(* CODESYS project plc_chalet_xts.library
   Title: CHALET_Xts
   Version: 1.7.6
   Placeholder: CHALET_Xts
   Company: Beckhoff CH

Project tree, tasks and I/O mapping:
  libraries: CHALET_BaseComponents, * (Beckhoff CH); CHALET_Nc, * (Beckhoff CH); Tc2_EtherCAT, * (Beckhoff Automation GmbH); Tc2_Math, * (Beckhoff Automation GmbH); Tc2_MC2, * (Beckhoff Automation GmbH); Tc2_Standard, * (Beckhoff Automation GmbH); Tc2_System, * (Beckhoff Automation GmbH); Tc3_Mc3Definitions, * (Beckhoff Automation GmbH); Tc3_McCollisionAvoidance, * (Beckhoff Automation GmbH); Tc3_McCoordinatedMotion, * (Beckhoff Automation GmbH); Tc3_Module, * (Beckhoff Automation GmbH); Tc3_XTS_Utility, * (Beckhoff Automation GmbH)
  COMPENENTs/
    Casting/
      function ToEnvironment [ST]
      function ToGroup [ST]
      function ToMover [ST]
      function ToMover_PLC [ST]
      function ToStation [ST]
      function ToStation_PLC [ST]
      function ToTrigger [ST]
    Environment/
      function block FB_XTS_Environment [ST]: FB_init, HR, Initialize, TrackIsRing, TrackLength, Update, UtilityEnvirement
      interface I_XTS_Environment: HR, Initialize, TrackIsRing, TrackLength, Update, UtilityEnvirement
    Group/
      data type E_NcGroupCommands
      function block FB_XTS_Group [ST]: AddAxisListToGroup, AddingAxisToGroup, AllAxesStanding, ChangeGapMode, Disable, Enable, FB_init, GroupEnabled, HR, Initialize, OID, RemoveAxisFromGroup, Reset, UngroupAllAxes, Update, UtilityCAGroup
      interface I_XTS_Group: AddAxisListToGroup, AddingAxisToGroup, AllAxesStanding, ChangeGapMode, Disable, Enable, GroupEnabled, HR, Initialize, RemoveAxisFromGroup, Reset, UngroupAllAxes, Update, UtilityCAGroup
    Mover/
      function block FB_XTS_Axis [ST]: HaltCA, MoveAbsoluteCA, Update
      function block FB_XTS_Mover [ST]: Disable, Enable, HaltCA, MoveAbsCA, Reset, Coupled, DrivenDistance, Feedback, Gap, getAxisRef, IdentInGroup, LagDistance, MoveAbsPosition, MoveAbsVelocity, MoverInGroup, Moving, NextMover, OID, ParentStation, PositionOnTrack, SetAcceleration, SetVelocity, TargedStation, FB_init, Initialize, Update, UtilityMover
      interface I_XTS_Mover: Coupled, Disable, DrivenDistance, Enable, Feedback, Gap, getAxisRef, HaltCA, IdentInGroup, LagDistance, MoveAbsCA, MoveAbsPosition, MoveAbsVelocity, MoverInGroup, Moving, NextMover, OID, ParentStation, PositionOnTrack, Reset, SetAcceleration, SetVelocity, TargedStation, UtilityMover
      interface I_XTS_Mover_PLC: DrivenDistance, Gap, LagDistance, PositionOnTrack, SetVelocity, TargedStation, UtilityMover
    Station/
      data type E_Colors_ARGB
      function block FB_XTS_Station [ST]: AddMoverToQueue, AreMoversInPlace, CtsEmptySpaceInQueue, CtsMoversInQueue, DeleteMoversQueue, FB_init, HR, Initialize, LUID, MoverGapAtExit, MoverQueueSize, MoversInQueue, MoverVelocityAtExit, OID, PositionOnTrack, SendMoversToStation, StationBehinde, StationGroupID, StationInFront, SuppressDynamicsChange, TrySendMoverToNextStation, Update, UtilityStationInfo
      interface I_XTS_Station: AddMoverToQueue, AreMoversInPlace, CtsEmptySpaceInQueue, CtsMoversInQueue, DeleteMoversQueue, HR, MoverGapAtExit, MoverQueueSize, MoversInQueue, MoverVelocityAtExit, PositionOnTrack, SendMoversToStation, StationGroupID, StationInFront
      interface I_XTS_Station_PLC: AreMoversInPlace, MoverQueueSize, MoversInQueue, SendMoversToStation, SuppressDynamicsChange
    System/
      function block FB_XTS_System [ST]: Disable, Disabled, Disabling, Enable, Enabled, Enabling, Environment, Feedback, getMoverInFront, getStationInFront, Initialize, Initialized, LinkEnvironment, LinkGroup, Movers, RegisterMover, RegisterStation, RegisterTrigger, RegisterZone, Reset, Station, Stations, SuppressAllDynamicsChanges, TrackLength, Update
      interface I_XTS_System_PLC: Disable, Disabled, Enable, Enabled, Feedback, Initialize, Initialized, Reset, Station, SuppressAllDynamicsChanges, TrackLength, Update
      interface I_XTS_System_Registration: Disabled, Enabled, Environment, getMoverInFront, getStationInFront, Initialized, LinkEnvironment, LinkGroup, Movers, RegisterMover, RegisterStation, RegisterTrigger, RegisterZone, Stations, TrackLength
    Trigger/
      function block FB_XTS_Trigger [ST]: FB_init, HR, Initialize, ListOfMoversToCheck, MoverAtTrigger, MoverDetected, PositionOnTrack, Prepare, TimeStamp, TriggerDirection, Update
      interface I_XTS_Trigger: HR, ListOfMoversToCheck, MoverAtTrigger, MoverDetected, PositionOnTrack, TimeStamp, TriggerDirection
    Zone/
      function block FB_XTS_Zone [ST]: CtsMoversInZone, EndPositionOnTrack, FB_init, HR, Initialize, ListOfMoversToCheck, MoversInZone, Prepare, StartPositionOnTrack, Update
      interface I_XTS_Zone: CtsMoversInZone, EndPositionOnTrack, HR, ListOfMoversToCheck, MoversInZone, StartPositionOnTrack
    Class Diagram
  FUNCTIONs/
    function FUN_BuildLogString [ST]
    function FUN_GetDistToPosModulo [ST]
    function FUN_InLimitTest [ST]
  00000000-0000-0000-0000-000000000000|Disclaimer Standard DE R1006.pdf
  Disclaimer Standard DE R1006.pdf
  global variables XtsParameterlist
*)

// COMPENENTs/Group/E_NcGroupCommands
{attribute 'qualified_only'}
{attribute 'strict'}
{attribute 'to_string'}
TYPE E_NcGroupCommands :
(
	None:=0,
	GroupDisable:=150,
	GroupEnable,
	GroupReset,
	AddAxisListToGroup,
	RemoveAxisFromGroup,
	UngroupAllAxes
);
END_TYPE

// COMPENENTs/Station/E_Colors_ARGB
{attribute 'qualified_only'}
{attribute 'strict'}
{attribute 'to_string'}
TYPE E_Colors_ARGB : (
        Darkred              := 16#FF8B0000, // rgb(139,0,0)
        Brown                := 16#FFA52A2A, // rgb(165,42,42)
        Firebrick            := 16#FFB22222, // rgb(178,34,34)
        Crimson              := 16#FFDC143C, // rgb(220,20,60)
        Red                  := 16#FFFF0000, // rgb(255,0,0)
        Tomato               := 16#FFFF6347, // rgb(255,99,71)
        Coral                := 16#FFFF7F50, // rgb(255,127,80)
        Indianred            := 16#FFCD5C5C, // rgb(205,92,92)
        Lightcoral           := 16#FFF08080, // rgb(240,128,128)
        Darksalmon           := 16#FFE9967A, // rgb(233,150,122)
        Salmon               := 16#FFFA8072, // rgb(250,128,114)
        Lightsalmon          := 16#FFFFA07A, // rgb(255,160,122)
        Orangered            := 16#FFFF4500, // rgb(255,69,0)
        Darkorange           := 16#FFFF8C00, // rgb(255,140,0)
        Orange               := 16#FFFFA500, // rgb(255,165,0)
        Gold                 := 16#FFFFD700, // rgb(255,215,0)
        Darkgoldenrod        := 16#FFB8860B, // rgb(184,134,11)
        Goldenrod            := 16#FFDAA520, // rgb(218,165,32)
        Palegoldenrod        := 16#FFEEE8AA, // rgb(238,232,170)
        Darkkhaki            := 16#FFBDB76B, // rgb(189,183,107)
        Khaki                := 16#FFF0E68C, // rgb(240,230,140)
        Olive                := 16#FF808000, // rgb(128,128,0)
        Yellow               := 16#FFFFFF00, // rgb(255,255,0)
        Yellowgreen          := 16#FF9ACD32, // rgb(154,205,50)
        Darkolivegreen       := 16#FF556B2F, // rgb(85,107,47)
        Olivedrab            := 16#FF6B8E23, // rgb(107,142,35)
        Lawngreen            := 16#FF7CFC00, // rgb(124,252,0)
        Chartreuse           := 16#FF7FFF00, // rgb(127,255,0)
        Greenyellow          := 16#FFADFF2F, // rgb(173,255,47)
        Darkgreen            := 16#FF006400, // rgb(0,100,0)
        Green                := 16#FF008000, // rgb(0,128,0)
        Forestgreen          := 16#FF228B22, // rgb(34,139,34)
        Lime                 := 16#FF00FF00, // rgb(0,255,0)
        Limegreen            := 16#FF32CD32, // rgb(50,205,50)
        Lightgreen           := 16#FF90EE90, // rgb(144,238,144)
        Palegreen            := 16#FF98FB98, // rgb(152,251,152)
        Darkseagreen         := 16#FF8FBC8F, // rgb(143,188,143)
        Mediumspringgreen    := 16#FF00FA9A, // rgb(0,250,154)
        Springgreen          := 16#FF00FF7F, // rgb(0,255,127)
        Seagreen             := 16#FF2E8B57, // rgb(46,139,87)
        Mediumaquamarine     := 16#FF66CDAA, // rgb(102,205,170)
        Mediumseagreen       := 16#FF3CB371, // rgb(60,179,113)
        Lightseagreen        := 16#FF20B2AA, // rgb(32,178,170)
        Darkslategray        := 16#FF2F4F4F, // rgb(47,79,79)
        Teal                 := 16#FF008080, // rgb(0,128,128)
        Darkcyan             := 16#FF008B8B, // rgb(0,139,139)
        Aqua                 := 16#FF00FFFF, // rgb(0,255,255)
        Lightcyan            := 16#FFE0FFFF, // rgb(224,255,255)
        Darkturquoise        := 16#FF00CED1, // rgb(0,206,209)
        Turquoise            := 16#FF40E0D0, // rgb(64,224,208)
        Mediumturquoise      := 16#FF48D1CC, // rgb(72,209,204)
        Paleturquoise        := 16#FFAFEEEE, // rgb(175,238,238)
        Aquamarine           := 16#FF7FFFD4, // rgb(127,255,212)
        Powderblue           := 16#FFB0E0E6, // rgb(176,224,230)
        Cadetblue            := 16#FF5F9EA0, // rgb(95,158,160)
        Steelblue            := 16#FF4682B4, // rgb(70,130,180)
        Cornflowerblue       := 16#FF6495ED, // rgb(100,149,237)
        Deepskyblue          := 16#FF00BFFF, // rgb(0,191,255)
        Dodgerblue           := 16#FF1E90FF, // rgb(30,144,255)
        Lightblue            := 16#FFADD8E6, // rgb(173,216,230)
        Skyblue              := 16#FF87CEEB, // rgb(135,206,235)
        Lightskyblue         := 16#FF87CEFA, // rgb(135,206,250)
        Midnightblue         := 16#FF191970, // rgb(25,25,112)
        Navy                 := 16#FF000080, // rgb(0,0,128)
        Darkblue             := 16#FF00008B, // rgb(0,0,139)
        Mediumblue           := 16#FF0000CD, // rgb(0,0,205)
        Blue                 := 16#FF0000FF, // rgb(0,0,255)
        Royalblue            := 16#FF4169E1, // rgb(65,105,225)
        Blueviolet           := 16#FF8A2BE2, // rgb(138,43,226)
        Indigo               := 16#FF4B0082, // rgb(75,0,130)
        Darkslateblue        := 16#FF483D8B, // rgb(72,61,139)
        Slateblue            := 16#FF6A5ACD, // rgb(106,90,205)
        Mediumslateblue      := 16#FF7B68EE, // rgb(123,104,238)
        Mediumpurple         := 16#FF9370DB, // rgb(147,112,219)
        Darkmagenta          := 16#FF8B008B, // rgb(139,0,139)
        Darkviolet           := 16#FF9400D3, // rgb(148,0,211)
        Darkorchid           := 16#FF9932CC, // rgb(153,50,204)
        Mediumorchid         := 16#FFBA55D3, // rgb(186,85,211)
        Purple               := 16#FF800080, // rgb(128,0,128)
        Thistle              := 16#FFD8BFD8, // rgb(216,191,216)
        Plum                 := 16#FFDDA0DD, // rgb(221,160,221)
        Violet               := 16#FFEE82EE, // rgb(238,130,238)
        Magenta              := 16#FFFF00FF, // rgb(255,0,255)
        Orchid               := 16#FFDA70D6, // rgb(218,112,214)
        Mediumvioletred      := 16#FFC71585, // rgb(199,21,133)
        Palevioletred        := 16#FFDB7093, // rgb(219,112,147)
        Deeppink             := 16#FFFF1493, // rgb(255,20,147)
        Hotpink              := 16#FFFF69B4, // rgb(255,105,180)
        Lightpink            := 16#FFFFB6C1, // rgb(255,182,193)
        Pink                 := 16#FFFFC0CB, // rgb(255,192,203)
        Antiquewhite         := 16#FFFAEBD7, // rgb(250,235,215)
        Beige                := 16#FFF5F5DC, // rgb(245,245,220)
        Bisque               := 16#FFFFE4C4, // rgb(255,228,196)
        Blanchedalmond       := 16#FFFFEBCD, // rgb(255,235,205)
        Wheat                := 16#FFF5DEB3, // rgb(245,222,179)
        Cornsilk             := 16#FFFFF8DC, // rgb(255,248,220)
        Lemonchiffon         := 16#FFFFFACD, // rgb(255,250,205)
        LightGoldenRodYellow := 16#FFFAFAD2, // rgb(250,250,210)
        LightYellow          := 16#FFFFFFE0, // rgb(255,255,224)
        SaddleBrown          := 16#FF8B4513, // rgb(139,69,19)
        Sienna               := 16#FFA0522D, // rgb(160,82,45)
        Chocolate            := 16#FFD2691E, // rgb(210,105,30)
        Peru                 := 16#FFCD853F, // rgb(205,133,63)
        SandyBrown           := 16#FFF4A460, // rgb(244,164,96)
        BurlyWood            := 16#FFDEB887, // rgb(222,184,135)
        RosyBrown            := 16#FFBC8F8F, // rgb(188,143,143)
        Moccasin             := 16#FFFFE4B5, // rgb(255,228,181)
        NavajoWhite          := 16#FFFFDEAD, // rgb(255,222,173)
        PeachPuff            := 16#FFFFDAB9, // rgb(255,218,185)
        MistyRose            := 16#FFFFE4E1, // rgb(255,228,225)
        LavenderBlush        := 16#FFFFF0F5, // rgb(255,240,245)
        Linen                := 16#FFFAF0E6, // rgb(250,240,230)
        OldLace              := 16#FFFDF5E6, // rgb(253,245,230)
        PapayaWhip           := 16#FFFFEFD5, // rgb(255,239,213)
        Seashell             := 16#FFFFF5EE, // rgb(255,245,238)
        MintCream            := 16#FFF5FFFA, // rgb(245,255,250)
        SlateGray            := 16#FF708090, // rgb(112,128,144)
        LightSlateGray       := 16#FF778899, // rgb(119,136,153)
        LightSteelBlue       := 16#FFB0C4DE, // rgb(176,196,222)
        Lavender             := 16#FFE6E6FA, // rgb(230,230,250)
        FloralWhite          := 16#FFFFFAF0, // rgb(255,250,240)
        AliceBlue            := 16#FFF0F8FF, // rgb(240,248,255)
        GhostWhite           := 16#FFF8F8FF, // rgb(248,248,255)
        HoneyDew             := 16#FFF0FFF0, // rgb(240,255,240)
        Ivory                := 16#FFFFFFF0, // rgb(255,255,240)
        Azure                := 16#FFF0FFFF, // rgb(240,255,255)
        Snow                 := 16#FFFFFAFA, // rgb(255,250,250)
        Black                := 16#FF000000, // rgb(0,0,0)
        DimGray              := 16#FF696969, // rgb(105,105,105)
        Gray                 := 16#FF808080, // rgb(128,128,128)
        DarkGray             := 16#FFA9A9A9, // rgb(169,169,169)
        Silver               := 16#FFC0C0C0, // rgb(192,192,192)
        LightGray            := 16#FFD3D3D3, // rgb(211,211,211)
        Gainsboro            := 16#FFDCDCDC, // rgb(220,220,220)
        WhiteSmoke           := 16#FFF5F5F5, // rgb(245,245,245)
        White                := 16#FFFFFFFF  // rgb(255,255,255)
    ) UDINT;
END_TYPE

// XtsParameterlist
{attribute 'qualified_only'}
VAR_GLOBAL CONSTANT
	MAX_MOVER_PER_SYSTEM : UINT := 50;
END_VAR

// COMPENENTs/Casting/ToEnvironment
FUNCTION ToEnvironment : BOOL
VAR_INPUT
	iChObject : I_CH_OBJECT;
	iXtsEnvironment : REFERENCE TO I_XTS_Environment;
END_VAR

VAR
	iTmp : I_XTS_Environment;
END_VAR

(* 
   1. Test if the interface exists
   2. Test if the object implements a "Object" interface 
   3. Write reference to interface in parameter
   4. Returne TRUE if succesfull
*)
IF iChObject <> 0 AND_THEN __QUERYINTERFACE(iChObject,iTmp) THEN
	iXtsEnvironment := iTmp;
	ToEnvironment := TRUE;
END_IF

END_FUNCTION

// COMPENENTs/Environment/I_XTS_Environment
INTERFACE I_XTS_Environment  EXTENDS __SYSTEM.IQueryInterface

{attribute 'monitoring':='call'}
PROPERTY HR : HRESULT
GET
END_GET
END_PROPERTY

METHOD Initialize : HRESULT
END_METHOD

{attribute 'monitoring':='call'}
PROPERTY TrackIsRing : BOOL
GET
END_GET
END_PROPERTY

{attribute 'monitoring':='call'}
PROPERTY TrackLength : LREAL
GET
END_GET
END_PROPERTY

METHOD Update : HRESULT
VAR_INPUT
END_VAR
END_METHOD

PROPERTY UtilityEnvirement : Tc3_XTS_Utility.i_TcIoXtsEnvironment
GET
END_GET
END_PROPERTY

END_INTERFACE

// COMPENENTs/Casting/ToGroup
FUNCTION ToGroup : BOOL
VAR_INPUT
	iChObject : I_CH_OBJECT;
	iXtsGroup : REFERENCE TO I_XTS_Group;
END_VAR

VAR
	iTmp : I_XTS_Group;
END_VAR

(* 
   1. Test if the interface exists
   2. Test if the object implements a "Object" interface 
   3. Write reference to interface in parameter
   4. Returne TRUE if succesfull
*)
IF iChObject <> 0 AND_THEN __QUERYINTERFACE(iChObject,iTmp) THEN
	iXtsGroup := iTmp;
	ToGroup := TRUE;
END_IF

END_FUNCTION

// COMPENENTs/Group/I_XTS_Group
INTERFACE I_XTS_Group  EXTENDS __SYSTEM.IQueryInterface

METHOD AddAxisListToGroup : HRESULT
VAR_INPUT
	iMovers : I_CH_List;
END_VAR
END_METHOD

METHOD AddingAxisToGroup : HRESULT
END_METHOD

PROPERTY AllAxesStanding : Bool
GET
END_GET
END_PROPERTY

METHOD ChangeGapMode : HRESULT
VAR_INPUT
	bFast : BOOL;
END_VAR
END_METHOD

METHOD Disable : HRESULT
VAR_INPUT
END_VAR
END_METHOD

METHOD Enable : HRESULT
VAR_INPUT
END_VAR
END_METHOD

{attribute 'monitoring':='call'}
PROPERTY GroupEnabled : BOOL
GET
END_GET
END_PROPERTY

{attribute 'monitoring':='call'}
PROPERTY HR : HRESULT
GET
END_GET
END_PROPERTY

METHOD Initialize : HRESULT
VAR_INPUT
END_VAR
END_METHOD

METHOD RemoveAxisFromGroup : HRESULT
VAR_INPUT
	iMover : I_XTS_Mover;
END_VAR
END_METHOD

METHOD Reset : HRESULT
VAR_INPUT
END_VAR
END_METHOD

METHOD UngroupAllAxes : HRESULT
VAR_INPUT
END_VAR
END_METHOD

METHOD Update : HRESULT
VAR_INPUT
END_VAR
END_METHOD

{attribute 'monitoring':='call'}
PROPERTY UtilityCAGroup : I_Mc2CaGroup
GET
END_GET
END_PROPERTY

END_INTERFACE

// COMPENENTs/Mover/I_XTS_Mover
INTERFACE I_XTS_Mover EXTENDS __SYSTEM.IQueryInterface

{attribute 'OPC.UA.DA.Property' := '1'}
{attribute 'monitoring':='call'}
PROPERTY Coupled : BOOL
GET
END_GET
END_PROPERTY

METHOD Disable : HRESULT
VAR_INPUT
END_VAR
END_METHOD

{attribute 'monitoring':='call'}
PROPERTY DrivenDistance : LREAL
GET
END_GET
END_PROPERTY

METHOD Enable : HRESULT
VAR_INPUT
END_VAR
END_METHOD

{attribute 'OPC.UA.DA.Property' := '1'}
{attribute 'monitoring':='call'}
PROPERTY Feedback : I_CH_Feedback
GET
END_GET
END_PROPERTY

{attribute 'monitoring':='call'}
PROPERTY Gap : LREAL
GET
END_GET
END_PROPERTY

PROPERTY getAxisRef : REFERENCE TO Tc2_MC2.AXIS_REF
GET
END_GET
END_PROPERTY

METHOD HaltCA : HRESULT
VAR_INPUT
END_VAR
END_METHOD

{attribute 'monitoring':='call'}
PROPERTY IdentInGroup : IDENT_IN_GROUP_REF
GET
END_GET
END_PROPERTY

{attribute 'monitoring':='call'}
PROPERTY LagDistance : LREAL
GET
END_GET
END_PROPERTY

METHOD MoveAbsCA : HRESULT
VAR_INPUT
    Position              : MC_LREAL := MC_INVALID;
    Velocity              : MC_LREAL := MC_INVALID;
    Gap                   : MC_LREAL := MC_DEFAULT;
    Direction             : Tc3_Mc3Definitions.MC_DIRECTION;
END_VAR
END_METHOD

{attribute 'monitoring':='call'}
PROPERTY MoveAbsPosition : LREAL
GET
END_GET
END_PROPERTY

{attribute 'monitoring':='call'}
PROPERTY MoveAbsVelocity : LREAL
GET
END_GET
END_PROPERTY

PROPERTY MoverInGroup : Bool
GET
END_GET
SET
END_SET
END_PROPERTY

{attribute 'OPC.UA.DA.Property' := '1'}
{attribute 'monitoring':='call'}
PROPERTY Moving : BOOL
GET
END_GET
END_PROPERTY

{attribute 'monitoring':='call'}
PROPERTY NextMover : I_XTS_Mover
GET
END_GET
END_PROPERTY

PROPERTY OID : OTCID
GET
END_GET
END_PROPERTY

{attribute 'monitoring':='call'}
PROPERTY ParentStation : I_XTS_Station
GET
END_GET
SET
END_SET
END_PROPERTY

{attribute 'monitoring':='call'}
PROPERTY PositionOnTrack : LREAL
GET
END_GET
END_PROPERTY

METHOD Reset : HRESULT
VAR_INPUT
END_VAR
END_METHOD

{attribute 'monitoring':='call'}
PROPERTY SetAcceleration : LREAL
GET
END_GET
END_PROPERTY

{attribute 'monitoring':='call'}
PROPERTY SetVelocity : LREAL
GET
END_GET
END_PROPERTY

{attribute 'monitoring':='call'}
PROPERTY TargedStation : STRING
GET
END_GET
SET
END_SET
END_PROPERTY

{attribute 'monitoring':='call'}
PROPERTY UtilityMover : I_TcIoXtsXpuMover
GET
END_GET
END_PROPERTY

END_INTERFACE

// COMPENENTs/Station/I_XTS_Station
INTERFACE I_XTS_Station  EXTENDS __SYSTEM.IQueryInterface

METHOD AddMoverToQueue : HRESULT
VAR_INPUT
	iMover : I_XTS_Mover;
END_VAR
END_METHOD

{attribute 'monitoring':='call'}
PROPERTY AreMoversInPlace : BOOL
GET
END_GET
END_PROPERTY

{attribute 'monitoring':='call'}
PROPERTY CtsEmptySpaceInQueue : UINT
GET
END_GET
END_PROPERTY

{attribute 'monitoring':='call'}
PROPERTY CtsMoversInQueue : UINT
GET
END_GET
END_PROPERTY

METHOD DeleteMoversQueue : HRESULT
VAR_INPUT
END_VAR
END_METHOD

{attribute 'monitoring':='call'}
PROPERTY HR : HRESULT
GET
END_GET
END_PROPERTY

{attribute 'monitoring':='call'}
PROPERTY MoverGapAtExit : LREAL
GET
END_GET
END_PROPERTY

{attribute 'monitoring':='call'}
PROPERTY MoverQueueSize : UINT
GET
END_GET
SET
END_SET
END_PROPERTY

{attribute 'monitoring':='call'}
PROPERTY MoversInQueue : REFERENCE TO ARRAY [0..(XtsParameterlist.MAX_MOVER_PER_SYSTEM-1)] OF I_XTS_Mover_PLC // Return a sorted list of movers in this zone. Index 0 is the mover in Front.
GET
END_GET
END_PROPERTY

{attribute 'monitoring':='call'}
PROPERTY MoverVelocityAtExit : LREAL
GET
END_GET
SET
END_SET
END_PROPERTY

{attribute 'monitoring':='call'}
PROPERTY PositionOnTrack : LREAL
GET
END_GET
END_PROPERTY

METHOD SendMoversToStation : HRESULT
VAR_INPUT
	TargedStation : STRING;
END_VAR
END_METHOD

{attribute 'monitoring':='call'}
PROPERTY StationGroupID : String
GET
END_GET
END_PROPERTY

{attribute 'monitoring':='call'}
PROPERTY StationInFront : I_XTS_Station
GET
END_GET
END_PROPERTY

END_INTERFACE

// COMPENENTs/Mover/I_XTS_Mover_PLC
INTERFACE I_XTS_Mover_PLC EXTENDS __SYSTEM.IQueryInterface

{attribute 'monitoring':='call'}
PROPERTY DrivenDistance : LREAL
GET
END_GET
END_PROPERTY

{attribute 'monitoring':='call'}
PROPERTY Gap : LREAL
GET
END_GET
END_PROPERTY

{attribute 'monitoring':='call'}
PROPERTY LagDistance : LREAL
GET
END_GET
END_PROPERTY

{attribute 'monitoring':='call'}
PROPERTY PositionOnTrack : LREAL
GET
END_GET
END_PROPERTY

{attribute 'monitoring':='call'}
PROPERTY SetVelocity : LREAL
GET
END_GET
END_PROPERTY

{attribute 'monitoring':='call'}
PROPERTY TargedStation : STRING
GET
END_GET
END_PROPERTY

{attribute 'monitoring':='call'}
PROPERTY UtilityMover : I_TcIoXtsXpuMover
GET
END_GET
END_PROPERTY

END_INTERFACE

// COMPENENTs/Casting/ToMover
FUNCTION ToMover : BOOL
VAR_INPUT
	iChObject : I_CH_OBJECT;
	iXtsMover : REFERENCE TO I_XTS_Mover;
END_VAR

VAR
	iTmp : I_XTS_Mover;
END_VAR

(* 
   1. Test if the interface exists
   2. Test if the object implements a "Object" interface 
   3. Write reference to interface in parameter
   4. Returne TRUE if succesfull
*)
IF iChObject <> 0 AND_THEN __QUERYINTERFACE(iChObject,iTmp) THEN
	iXtsMover := iTmp;
	ToMover := TRUE;
END_IF

END_FUNCTION

// COMPENENTs/Casting/ToMover_PLC
FUNCTION ToMover_PLC : BOOL
VAR_INPUT
	iChObject : I_CH_OBJECT;
	iXtsMover : REFERENCE TO I_XTS_Mover_PLC;
END_VAR

VAR
	iTmp : I_XTS_Mover_PLC;
END_VAR

(* 
   1. Test if the interface exists
   2. Test if the object implements a "Object" interface 
   3. Write reference to interface in parameter
   4. Returne TRUE if succesfull
*)
IF iChObject <> 0 AND_THEN __QUERYINTERFACE(iChObject,iTmp) THEN
	iXtsMover := iTmp;
	ToMover_PLC := TRUE;
END_IF

END_FUNCTION

// COMPENENTs/Casting/ToStation
FUNCTION ToStation : BOOL
VAR_INPUT
	iChObject : I_CH_OBJECT;
	iXtsStation : REFERENCE TO I_XTS_Station;
END_VAR

VAR
	iTmp : I_XTS_Station;
END_VAR

(* Register the Station
   1. Test if the interface exists
   2. Test if the object implements a "Object" interface 
*)
IF iChObject <> 0 AND_THEN __QUERYINTERFACE(iChObject,iTmp) THEN
	iXtsStation := iTmp;
	ToStation := TRUE;
END_IF

END_FUNCTION

// COMPENENTs/Casting/ToStation_PLC
FUNCTION ToStation_PLC : BOOL
VAR_INPUT
	iChObject : I_CH_OBJECT;
	iXtsStationPLC : REFERENCE TO I_XTS_Station_PLC;
END_VAR

VAR
	iTmp : I_XTS_Station_PLC;
END_VAR

(* Register the Station
   1. Test if the interface exists
   2. Test if the object implements a "Object" interface 
*)
IF iChObject <> 0 AND_THEN __QUERYINTERFACE(iChObject,iTmp) THEN
	iXtsStationPLC := iTmp;
	ToStation_PLC := TRUE;
END_IF

END_FUNCTION

// COMPENENTs/Station/I_XTS_Station_PLC
INTERFACE I_XTS_Station_PLC

{attribute 'monitoring':='call'}
PROPERTY AreMoversInPlace : BOOL
GET
END_GET
END_PROPERTY

{attribute 'monitoring':='call'}
PROPERTY MoverQueueSize : UINT
GET
END_GET
SET
END_SET
END_PROPERTY

{attribute 'monitoring':='call'}
PROPERTY MoversInQueue : REFERENCE TO ARRAY [0..(XtsParameterlist.MAX_MOVER_PER_SYSTEM-1)] OF I_XTS_Mover_PLC // Return a sorted list of movers in this zone. Index 0 is the mover in Front.
GET
END_GET
END_PROPERTY

METHOD SendMoversToStation : HRESULT
VAR_INPUT
	TargedStation : STRING;
END_VAR
END_METHOD

{attribute 'monitoring':='call'}
PROPERTY SuppressDynamicsChange : BOOL
GET
END_GET
SET
END_SET
END_PROPERTY

END_INTERFACE

// COMPENENTs/Casting/ToTrigger
FUNCTION ToTrigger : BOOL
VAR_INPUT
	iChObject : I_CH_OBJECT;
	iXtsTrigger : REFERENCE TO I_XTS_Trigger;
END_VAR

VAR
	iTmp : I_XTS_Trigger;
END_VAR

(* 
   1. Test if the interface exists
   2. Test if the object implements a "Object" interface 
   3. Write reference to interface in parameter
   4. Returne TRUE if succesfull
*)
IF iChObject <> 0 AND_THEN __QUERYINTERFACE(iChObject,iTmp) THEN
	iXtsTrigger := iTmp;
	ToTrigger := TRUE;
END_IF

END_FUNCTION

// COMPENENTs/Trigger/I_XTS_Trigger
INTERFACE I_XTS_Trigger  EXTENDS __SYSTEM.IQueryInterface

{attribute 'monitoring':='call'}
PROPERTY HR : HRESULT
GET
END_GET
END_PROPERTY

PROPERTY ListOfMoversToCheck : I_CH_List
SET
END_SET
END_PROPERTY

{attribute 'monitoring':='call'}
PROPERTY MoverAtTrigger : I_XTS_Mover
GET
END_GET
END_PROPERTY

{attribute 'monitoring':='call'}
PROPERTY MoverDetected : BOOL
GET
END_GET
END_PROPERTY

{attribute 'monitoring':='call'}
PROPERTY PositionOnTrack : LREAL
GET
END_GET
SET
END_SET
END_PROPERTY

{attribute 'monitoring':='call'}
PROPERTY TimeStamp : T_DCTIME64;
GET
END_GET
END_PROPERTY

{attribute 'monitoring':='call'}
PROPERTY TriggerDirection : Tc2_MC2.MC_Direction
GET
END_GET
SET
END_SET
END_PROPERTY

END_INTERFACE

// COMPENENTs/Environment/FB_XTS_Environment
{attribute 'no_explicit_call' := 'Do not call the body - Stick to OOP'}
FUNCTION_BLOCK FB_XTS_Environment EXTENDS FB_CH_Object IMPLEMENTS I_XTS_Environment
VAR
	{attribute 'hide'}
	iXtsSystem : I_XTS_System_Registration;

	fbUtilityEnvironment : Tc3_XTS_Utility.FB_TcIoXtsEnvironment;
	
	{attribute 'hide'}
	fbXtsEnvironmentVisu : Tc3_XTS_Utility.FB_XtsEnvironmentVisu;
		
END_VAR

METHOD FB_init : BOOL
VAR_INPUT
	bInitRetains : BOOL; // if TRUE, the retain variables are initialized (warm start / cold start)
	bInCopyCode : BOOL;  // if TRUE, the instance afterwards gets moved into the copy code (online change)

	iXtsSystem : I_XTS_System_Registration; //Interface to XTS system object	
END_VAR
//Regristrate object in System
IF iXtsSystem <> 0 THEN
	iXtsSystem.LinkEnvironment(THIS^);
	THIS^.iXtsSystem := iXtsSystem;
END_IF
END_METHOD

{warning 'add property implementation'}
{attribute 'monitoring':='call'}
PROPERTY HR : HRESULT
GET
END_GET
END_PROPERTY

METHOD Initialize : HRESULT
VAR_INST
	bInitDone :BOOL := FALSE;
END_VAR
IF NOT bInitDone THEN
	Initialize := S_PENDING;	

	//Enable init Info Server if needed
	fbUtilityEnvironment.P_XtsEnvironmentConfiguration.bEnableInitInfoServer := TRUE;

	//Enable init CA Group if needed
	fbUtilityEnvironment.P_XtsEnvironmentConfiguration.bEnableInitCaGroup := TRUE;

	//Start init
	IF fbUtilityEnvironment.Init(bExecute := TRUE) THEN
		//Stop init
		fbUtilityEnvironment.Init(bExecute := FALSE);
		bInitDone := TRUE;
	END_IF
	
	// Link data Pointer 
	fbXtsEnvironmentVisu(ipTcIoXtsEnvironment:=UtilityEnvirement);
ELSE
	//Check if init succeeded
	IF fbUtilityEnvironment.P_IsInitialized THEN
		// check if the position detection of the Movers has been completed
		IF NOT fbUtilityEnvironment.XpuTcIo(1).GetAreAllPositionsValid()
		OR NOT fbUtilityEnvironment.XpuTcIo(1).GetIsTeachingValid()
		OR NOT fbUtilityEnvironment.XpuTcIo(1).GetDetectedMoverCount() = fbUtilityEnvironment.XpuTcIo(1).GetExpectedMoverCount() THEN
			Initialize := S_OK;		
		END_IF
	END_IF
END_IF
END_METHOD

{attribute 'monitoring':='call'}
PROPERTY TrackIsRing : BOOL
GET
IF fbUtilityEnvironment.P_IsInitialized THEN
	TrackIsRing := fbUtilityEnvironment.Mc2CaGroup(1).GetRailIsRing();
END_IF
END_GET
END_PROPERTY

{attribute 'monitoring':='call'}
PROPERTY TrackLength : LREAL
GET
IF fbUtilityEnvironment.P_IsInitialized THEN
	TrackLength := fbUtilityEnvironment.Mc2CaGroup(1).GetRailLength();
END_IF
END_GET
END_PROPERTY

METHOD Update : HRESULT
VAR_INPUT
END_VAR
VAR
	hr : HRESULT;
END_VAR
hr := S_OK;

fbXtsEnvironmentVisu.Cycle();

Update:= hr;
END_METHOD

PROPERTY UtilityEnvirement : Tc3_XTS_Utility.i_TcIoXtsEnvironment
GET
UtilityEnvirement := fbUtilityEnvironment;
END_GET
END_PROPERTY

END_FUNCTION_BLOCK

// COMPENENTs/System/I_XTS_System_Registration
INTERFACE I_XTS_System_Registration

{attribute 'monitoring':='call'}
PROPERTY Disabled : Bool
GET
END_GET
END_PROPERTY

{attribute 'monitoring':='call'}
PROPERTY Enabled : Bool
GET
END_GET
END_PROPERTY

{attribute 'monitoring':='call'}
PROPERTY Environment : I_XTS_Environment
GET
END_GET
END_PROPERTY

METHOD getMoverInFront : I_Xts_Mover
VAR_INPUT
	iMover : I_Xts_Mover;
END_VAR
END_METHOD

METHOD getStationInFront : I_XTS_Station
VAR_INPUT
	iStation : I_XTS_Station;
END_VAR
END_METHOD

{attribute 'monitoring':='call'}
PROPERTY Initialized : BOOL
GET
END_GET
END_PROPERTY

METHOD LinkEnvironment : HRESULT
VAR_INPUT
	iEnvironment : I_CH_Object;
END_VAR
END_METHOD

METHOD LinkGroup : HRESULT
VAR_INPUT
	Group : I_CH_Object;
END_VAR
END_METHOD

{attribute 'monitoring':='call'}
PROPERTY Movers : CHALET_BaseComponents.I_CH_LIST
GET
END_GET
END_PROPERTY

METHOD RegisterMover : HRESULT
VAR_INPUT
	Mover : I_CH_Object;
END_VAR
END_METHOD

METHOD RegisterStation : HRESULT
VAR_INPUT
	Station : I_CH_Object;
END_VAR
END_METHOD

METHOD RegisterTrigger : HRESULT
VAR_INPUT
	Trigger	: CHALET_BaseComponents.I_CH_Object;
END_VAR
END_METHOD

METHOD RegisterZone : HRESULT
VAR_INPUT
	Zone	: CHALET_BaseComponents.I_CH_Object;
END_VAR
END_METHOD

PROPERTY Stations : I_CH_LIST
GET
END_GET
END_PROPERTY

{attribute 'monitoring':='call'}
PROPERTY TrackLength : LREAL
GET
END_GET
END_PROPERTY

END_INTERFACE

// COMPENENTs/Group/FB_XTS_Group
{attribute 'no_explicit_call' := 'Do not call the body - Stick to OOP'}
FUNCTION_BLOCK FB_XTS_Group EXTENDS FB_CH_Object IMPLEMENTS I_XTS_Group
VAR
	{attribute 'hide'}
	iXtsSystem : I_XTS_System_Registration;
	{attribute 'hide'}
	iUtilityCAGroup : I_Mc2CaGroup;
	{attribute 'hide'}
	fbAddAxisToGroup : Tc3_McCoordinatedMotion.MC_AddAxisToGroup;
	{attribute 'hide'}
	fbRemoveAxisToGroup : Tc3_McCoordinatedMotion.MC_RemoveAxisFromGroup;
	{attribute 'hide'}
	fbGroupEnable : Tc3_McCoordinatedMotion.MC_GroupEnable;
	{attribute 'hide'}
	fbGroupDisable : Tc3_McCoordinatedMotion.MC_GroupDisable;
	{attribute 'hide'}
	fbGroupReadStatus : Tc3_McCoordinatedMotion.MC_GroupReadStatus;	
	{attribute 'hide'}
	fbUngroupAllAxes : Tc3_McCoordinatedMotion.MC_UngroupAllAxes;	
	{attribute 'hide'}
	fbGroupReset : Tc3_McCoordinatedMotion.MC_GroupReset;
	{attribute 'hide'}
	nState_SEQ_Adding : UINT;
	{attribute 'hide'}	
	bInitDone : BOOL;
	{attribute 'hide'}	
	fbMovers : FB_CH_List; // List of Axis to be added to the group
		
	
	GroupRef : AXES_GROUP_REF;
	
	{attribute 'hide'}	
	iTempMover : I_XTS_Mover;

	{attribute 'hide'}
	dummyAxis : AXIS_REF;
	{attribute 'hide'}	
	fbFeedback : FB_CH_Feedback;
	{attribute 'hide'}
	_eActiveCommand 		: E_NcGroupCommands := E_NcGroupCommands.None;

END_VAR

METHOD AddAxisListToGroup : HRESULT
VAR_INPUT
	iMovers : I_CH_List;
END_VAR
IF NOT THIS^.fbFeedback.Done THEN
	//Errror active/not ready
	THIS^.fbFeedback.LastCommandAccepted := FALSE;
	
ELSIF nState_SEQ_Adding <> 0 AND nState_SEQ_Adding <> 999 THEN
	// Adding Sequence is not finished. Terminate first
	THIS^.fbFeedback.LastCommandAccepted := FALSE;

ELSIF iMovers = 0 THEN
	// Invalide input
	THIS^.fbFeedback.LastCommandAccepted := FALSE;
		
ELSE
	// duplicate List
	THIS^.fbMovers.Duplicate(CopyFrom := iMovers);
	
	
	THIS^.nState_SEQ_Adding := 1;
	THIS^.fbFeedback.LastCommandAccepted := TRUE;
	THIS^._eActiveCommand := E_NcGroupCommands.AddAxisListToGroup;
	THIS^.fbFeedback.Busy := TRUE;	

END_IF

IF THIS^.fbFeedback.LastCommandAccepted THEN
	AddAxisListToGroup := S_OK;
ELSE
	AddAxisListToGroup := E_FAIL;
END_IF
END_METHOD

METHOD AddingAxisToGroup : HRESULT
VAR
	hr : HRESULT;
END_VAR
VAR_INST
	iMover : I_CH_Object;
END_VAR
AddingAxisToGroup := S_PENDING;

CASE nState_SEQ_Adding OF
	0: // Idle
		AddingAxisToGroup := S_OK;
		
		
	1: // prepare List for iteratrion 
		THIS^.fbMovers.ResetIterator();
		nState_SEQ_Adding := 10;
		
		
	10: // has next Mover?
		IF THIS^.fbMovers.HasNextObject() THEN
			iMover := THIS^.fbMovers.GetNextObject();
			IF ToMover(iMover, iTempMover) THEN
				nState_SEQ_Adding := 20;
			END_IF
		ELSE 
			nState_SEQ_Adding := 100;			
		END_IF
		
		
	20: // get Axis Reference
		IF iTempMover <> 0 AND_THEN __ISVALIDREF(iTempMover.getAxisRef) THEN
			nState_SEQ_Adding := 30;
		END_IF
		
		
	30: // add mover to group
		fbAddAxisToGroup.Execute := TRUE;
		IF fbAddAxisToGroup.Error THEN
			nState_SEQ_Adding := 1000 + nState_SEQ_Adding;
		ELSIF fbAddAxisToGroup.Done THEN
			nState_SEQ_Adding := 40;
			iTempMover.MoverInGroup := TRUE;
		END_IF

	40: // Remove Object from List
		IF THIS^.fbMovers.RemoveObject(iMover) THEN
			THIS^.fbMovers.ResetIterator();
			nState_SEQ_Adding := 10;
		ELSE
			nState_SEQ_Adding := 1000 + nState_SEQ_Adding;	
		END_IF
			
		
	100: // clear list
		// todo THIS^.iMovers.Clear();	
		nState_SEQ_Adding := 999;
		
		
	999: // Done
		AddingAxisToGroup := S_OK;

		
	1000..1999://Error
		hr := GetMostSignificant(hr, E_FAIL);	
			
END_CASE

// Propagate error
IF FAILED(hr) THEN
	AddingAxisToGroup := hr;
END_IF

// set feedback
THIS^.fbFeedback.HR := hr;
END_METHOD

{warning 'Eigenschaftenimplementierung hinzufügen'}
PROPERTY AllAxesStanding : BOOL
GET
AllAxesStanding := fbGroupReadStatus.AllAxesStanding;
END_GET
END_PROPERTY

METHOD ChangeGapMode : HRESULT
VAR_INPUT
	bFast : BOOL;
END_VAR
VAR
	hr : HRESULT;
	iCaGroup: I_Mc2CaGroup;
END_VAR
ChangeGapMode := S_PENDING;

IF bFast THEN
	// Change fist to positive direction and then to Fast Mode	
	iUtilityCAGroup.SetGapControlDirection(MC_GAP_CONTROL_DIRECTION.mcGapCtrlDirectionPositive);
	iUtilityCAGroup.SetDefaultGapControlMode(MC_DEFAULT_GAP_CONTROL_MODE.mcGapCtrlModeFast);
ELSE
	// Change first to StandardMode and then to both direction
	iUtilityCAGroup.SetDefaultGapControlMode(MC_DEFAULT_GAP_CONTROL_MODE.mcGapCtrlModeStandard);
	iUtilityCAGroup.SetGapControlDirection(MC_GAP_CONTROL_DIRECTION.mcGapCtrlDirectionBoth);
END_IF

ChangeGapMode := S_OK;
END_METHOD

METHOD Disable : HRESULT
THIS^.fbFeedback.LastCommandAccepted := TRUE;
THIS^.fbFeedback.Busy := TRUE;	
THIS^.fbGroupDisable.Execute := TRUE;
THIS^._eActiveCommand := E_NcGroupCommands.GroupDisable;

Disable := S_OK;
END_METHOD

METHOD Enable : HRESULT
IF NOT THIS^.fbFeedback.Done THEN
	THIS^.fbFeedback.LastCommandAccepted := FALSE;
	// Error active/not ready
	
ELSIF NOT(THIS^.fbGroupReadStatus.GroupDisabled) THEN
	THIS^.fbFeedback.LastCommandAccepted := FALSE;
	// Group in wrong State
	
ELSE
	THIS^.fbFeedback.LastCommandAccepted := TRUE;
	THIS^.fbFeedback.Busy := TRUE;
	THIS^._eActiveCommand := E_NcGroupCommands.GroupEnable;
	THIS^.fbGroupEnable.Execute := TRUE;
END_IF

IF THIS^.fbFeedback.LastCommandAccepted THEN
	Enable := S_OK;
ELSE  
	Enable := E_FAIL;;	
END_IF
END_METHOD

METHOD FB_init : BOOL
VAR_INPUT
	bInitRetains : BOOL; // if TRUE, the retain variables are initialized (warm start / cold start)
	bInCopyCode : BOOL;  // if TRUE, the instance afterwards gets moved into the copy code (online change)
	
	iXtsSystem : I_XTS_System_Registration; //Interface to XTS system object	
END_VAR
//Regristrate object in System
IF iXtsSystem <> 0 THEN
	iXtsSystem.LinkGroup(THIS^);
	THIS^.iXtsSystem := iXtsSystem;
END_IF
END_METHOD

{attribute 'monitoring':='call'}
PROPERTY GroupEnabled : BOOL
GET
GroupEnabled := fbGroupReadStatus.Valid AND NOT (fbGroupReadStatus.GroupDisabled OR fbGroupReadStatus.GroupErrorStop);
END_GET
END_PROPERTY

{attribute 'monitoring':='call'}
PROPERTY HR : HRESULT
GET
HR := fbFeedback.hr;
END_GET
END_PROPERTY

METHOD Initialize : HRESULT
VAR_INPUT
END_VAR
IF NOT THIS^.bInitDone THEN

	Initialize := S_PENDING;

	
	// Check if link to Group is mapped
	IF NcParameterlist.ERROR_IF_NC_AXIS_IS_NOT_MAPPED AND_THEN F_GetMappingStatus(ADR(THIS^.GroupRef.NcToPlc), SIZEOF(THIS^.GroupRef.NcToPlc)) <> EPlcMappingStatus.MS_Mapped THEN
		//ERROR NcToPlc
		Initialize := E_FAIL;
		RETURN;
	END_IF
	
	
	// Check if link to Group is mapped
	IF NcParameterlist.ERROR_IF_NC_AXIS_IS_NOT_MAPPED AND_THEN F_GetMappingStatus(ADR(THIS^.GroupRef.PlcToNc), SIZEOF(THIS^.GroupRef.PlcToNc)) <> EPlcMappingStatus.MS_Mapped THEN
		//ERROR PlcToNc
		Initialize := E_FAIL;		
		RETURN;
	END_IF	


		
	IF THIS^.iXtsSystem.Environment <> 0 THEN
		iUtilityCAGroup := THIS^.iXtsSystem.Environment.UtilityEnvirement.Mc2CaGroup(1);
	END_IF

	THIS^.bInitDone := TRUE;
ELSE
	
	Initialize := S_OK;

END_IF
END_METHOD

{attribute 'monitoring':='call'}
PROPERTY OID : OTCID
GET
OID := GroupRef.NcToPlc.Common.GroupOID;
END_GET
END_PROPERTY

METHOD RemoveAxisFromGroup : HRESULT
VAR_INPUT
	iMover	: I_XTS_Mover;
END_VAR

VAR
	Axis : I_Adapter_AXIS_REF;
END_VAR
IF iMover <> 0 AND_THEN __QUERYINTERFACE(iMover, Axis) THEN
	
	THIS^._eActiveCommand := E_NcGroupCommands.RemoveAxisFromGroup;
	THIS^.fbFeedback.LastCommandAccepted := TRUE;
	THIS^.fbFeedback.Busy := TRUE;

	fbRemoveAxisToGroup.IdentInGroup := iMover.IdentInGroup;
	fbRemoveAxisToGroup.Execute := TRUE;
	iMover.MoverInGroup := FALSE;
	
	RemoveAxisFromGroup := S_OK;

ELSE
	THIS^.fbFeedback.LastCommandAccepted := FALSE;
END_IF
END_METHOD

METHOD Reset : HRESULT
THIS^._eActiveCommand := E_NcGroupCommands.GroupReset;
THIS^.fbFeedback.LastCommandAccepted := TRUE;
THIS^.fbFeedback.Busy := TRUE;	

THIS^.fbGroupReset.Execute := TRUE;

Reset := S_OK;
END_METHOD

METHOD UngroupAllAxes : HRESULT
THIS^._eActiveCommand := E_NcGroupCommands.UngroupAllAxes;
THIS^.fbFeedback.LastCommandAccepted := TRUE;
THIS^.fbFeedback.Busy := TRUE;	

THIS^.nState_SEQ_Adding := 0;

THIS^.fbUngroupAllAxes.Execute := TRUE;

UngroupAllAxes := S_OK;
END_METHOD

METHOD Update : HRESULT
// ********************** Refresh Group Information ***********************************************
fbGroupReadStatus(AxesGroup:=  THIS^.GroupRef, Enable:= TRUE);

// ********************** Set feedback depending on active command *******************************
IF THIS^._eActiveCommand <> E_NcGroupCommands.None THEN
	fbFeedback.ActiveCommand 	:= TO_STRING(THIS^._eActiveCommand);	
END_IF

CASE THIS^._eActiveCommand OF 
  E_NcGroupCommands.GroupDisable:
		fbFeedback.Busy 		:= fbGroupDisable.Busy;
		fbFeedback.Done 		:= fbGroupDisable.Done;
		fbFeedback.ErrorId 		:= fbGroupDisable.ErrorId;
  
  E_NcGroupCommands.GroupEnable:
		fbFeedback.Busy 		:= fbGroupEnable.Busy;
		fbFeedback.Done 		:= fbGroupEnable.Done;
		fbFeedback.ErrorId 		:= fbGroupEnable.ErrorId;
  
  E_NcGroupCommands.GroupReset:
		fbFeedback.Busy 		:= fbGroupReset.Busy;
		fbFeedback.Done 		:= fbGroupReset.Done;
		fbFeedback.ErrorId 		:= fbGroupReset.ErrorId;  
  
  E_NcGroupCommands.AddAxisListToGroup: 
		fbFeedback.Busy 		:= nState_SEQ_Adding > 0 AND nState_SEQ_Adding < 999;
		fbFeedback.Done 		:= nState_SEQ_Adding = 999; 
//		fbFeedback.ErrorId 		:= ;
  
  E_NcGroupCommands.RemoveAxisFromGroup:
		fbFeedback.Busy 		:= fbRemoveAxisToGroup.Busy;
		fbFeedback.Done 		:= fbRemoveAxisToGroup.Done;
		fbFeedback.ErrorId 		:= fbRemoveAxisToGroup.ErrorId;
  
  E_NcGroupCommands.UngroupAllAxes:
		fbFeedback.Busy 		:= fbUngroupAllAxes.Busy;
		fbFeedback.Done 		:= fbUngroupAllAxes.Done;
		fbFeedback.ErrorId 		:= fbUngroupAllAxes.ErrorId;
  
END_CASE

// **********************  Stop to execute commands on .done or .error ***************************
IF THIS^.fbFeedback.Done OR THIS^.fbFeedback.Error THEN
	THIS^._eActiveCommand 				:= E_NcGroupCommands.None;
END_IF


// **********************  Cyclic calls  *********************************************************
IF THIS^.iTempMover <> 0 THEN
	fbAddAxisToGroup(AxesGroup := THIS^.GroupRef, Axis := THIS^.iTempMover.getAxisRef, IdentInGroup := iTempMover.IdentInGroup);
ELSE
	fbAddAxisToGroup(AxesGroup := THIS^.GroupRef, Axis := dummyAxis);
END_IF

fbRemoveAxisToGroup(AxesGroup := THIS^.GroupRef);
fbGroupEnable(AxesGroup := THIS^.GroupRef);
fbGroupDisable(AxesGroup := THIS^.GroupRef);
fbUngroupAllAxes(AxesGroup := THIS^.GroupRef);
fbGroupReset(AxesGroup := THIS^.GroupRef);

// ********************** Reset all Execution flags **********************************************
fbAddAxisToGroup.Execute := FALSE;
fbRemoveAxisToGroup.Execute := FALSE;
fbGroupEnable.Execute := FALSE;
fbGroupDisable.Execute := FALSE;
fbUngroupAllAxes.Execute := FALSE;
fbGroupReset.Execute := FALSE;


// todo hresult
END_METHOD

{attribute 'monitoring':='call'}
PROPERTY UtilityCAGroup : I_Mc2CaGroup
GET
UtilityCAGroup := THIS^.iUtilityCAGroup;
END_GET
END_PROPERTY

END_FUNCTION_BLOCK

// COMPENENTs/Mover/FB_XTS_Axis
{attribute 'no_explicit_call' := 'Do not call the body - Stick to OOP'}
FUNCTION_BLOCK FB_XTS_Axis EXTENDS CHALET_NC.FB_NcAxis
VAR
	{attribute 'hide'}
	fbMoveAbsoluteCA		: ARRAY [0..1] OF MC_MoveAbsoluteCA;//A second function block is always required to use the BufferMode. It is not possible to trigger a move function block with new parameters while it is active.
	{attribute 'hide'}
	fbHaltCA				: MC_HaltCA;
	{attribute 'hide'}
	nActiveMoveAbsCa 		: UINT;
END_VAR

METHOD HaltCA : HRESULT
VAR_INPUT
	lrDeceleration          : LREAL;
    lrJerk                  : LREAL;
    lrGap                   : LREAL;
END_VAR
IF THIS^.Error THEN
	THIS^.fbFeedback.LastCommandAccepted	:= FALSE;
	//Error active/not ready
		
//ELSIF NOT(THIS^.Axis.Status.StandStill OR THIS^.Axis.Status.DiscreteMotion OR THIS^.Axis.Status.ContinuousMotion OR THIS^.Axis.Status.SynchronizedMotion) THEN		
//	THIS^.fbFeedback.LastCommandAccepted	:= FALSE;
//	//Axis in wrong State
		
ELSE
	THIS^.eActiveCommand 				:= E_NcAxisCommands.HaltCA;
	THIS^.fbFeedback.LastCommandAccepted:= TRUE;		
	THIS^.fbFeedback.Busy 				:= TRUE;
	
	THIS^.fbHaltCA.Execute		:= TRUE;
	THIS^.fbHaltCA.Gap			:= lrGap;
	
	
	//Deceleration
	//If input = 0  then use default dynamics
	IF lrDeceleration = 0.0 THEN
		THIS^.fbHaltCA.Deceleration := THIS^.lrDefaultDeceleration;
	ELSE
		THIS^.fbHaltCA.Deceleration := lrDeceleration;
	END_IF
	
	//Jerk
	//If input = 0  then use default dynamics
	IF lrJerk = 0.0 THEN
		THIS^.fbHaltCA.Jerk := THIS^.lrDefaultJerk;
	ELSE
		THIS^.fbHaltCA.Jerk := lrJerk;
	END_IF

END_IF


HaltCA := THIS^.fbFeedback.HR;
END_METHOD

{attribute 'TcRpcEnable':='1'} //call methode via OPC-UA conection
METHOD MoveAbsoluteCA  : I_CH_Feedback
VAR_INPUT
	lrPosition		: LREAL;
	
	(* Use the default dynamics if input=0. 
	The default dynamics can be read and written via property and is initialized with the default values in the NC parameter list. *)
	lrVelocity		: LREAL;
	
	(* This value determines the minimum gap to the predecessor for Collision Avoidance. If no value is entered, the default value of the group is used.*)
	lrGap		: LREAL;
	
	(* Defines the direction of the movement (e.g. for a modulo axis). *)
	Direction	: Tc3_Mc3Definitions.MC_DIRECTION;
	
	(* Use the default dynamics if input=0. 
	The default dynamics can be read and written via property and is initialized with the default values in the NC parameter list. *)
	lrAcceleration	: LREAL;
	
	(* Use the default dynamics if input=0. 
	The default dynamics can be read and written via property and is initialized with the default values in the NC parameter list. *)
	lrDeceleration	: LREAL;
	
	(* Use the default dynamics if input=0. 
	The default dynamics can be read and written via property and is initialized with the default values in the NC parameter list. *)
	lrJerk			: LREAL;
	

	(* Use the default mode without buffering if input=0. 
	BufferModes:
		-MC_Aborting: Default mode without buffering. The command is executed immediately and interrupts any other command that may be running.
		-MC_Buffered: The command is executed once no other command is running on the axis. The previous movement continues until it has stopped. The following command is started from standstill. *)
	BufferMode   : MC_BufferMode;
END_VAR
VAR
	nInactiveInstance : UINT;
END_VAR
IF THIS^.Error THEN
	THIS^.fbFeedback.LastCommandAccepted	:= FALSE;
	//Error active/not ready

ELSIF NOT THIS^.BufferEmpty THEN		
	THIS^.fbFeedback.LastCommandAccepted	:= FALSE;
	//Buffer not ready to store next motion command	
	
ELSIF NOT((BufferMode <> MC_BufferMode.MC_Aborting) OR (BufferMode <> MC_BufferMode.MC_Buffered)) THEN		
	THIS^.fbFeedback.LastCommandAccepted	:= FALSE;
	//only mcAborting and mcBuffered are available 	
	
ELSIF NOT(THIS^.Axis.Status.StandStill OR THIS^.Axis.Status.DiscreteMotion OR THIS^.Axis.Status.ContinuousMotion OR THIS^.Axis.Status.SynchronizedMotion) THEN		
	THIS^.fbFeedback.LastCommandAccepted	:= FALSE;
	//Axis in wrong State
	
ELSIF (BufferMode <> MC_BufferMode.MC_Aborting) AND bNewBufferCommadThisCycle THEN		
	THIS^.fbFeedback.LastCommandAccepted	:= FALSE;
	//Buffer not ready to store next motion command		
	//Max send one buffered motion command each cycle	
	
ELSE
	//A second function block is always required to use the BufferMode. It is not possible to trigger a move function block with new parameters while it is active.
	IF THIS^.fbMoveAbsoluteCA[nActiveMoveAbsCA].Busy THEN
		nInactiveInstance := (THIS^.nActiveMoveAbsCa + 1)MOD 2;
	ELSE
		nInactiveInstance := THIS^.nActiveMoveAbsCa;
	END_IF
	
	THIS^.eActiveCommand 				:= E_NcAxisCommands.MoveAbsoluteCA;
	THIS^.fbFeedback.LastCommandAccepted:= TRUE;		
	THIS^.fbFeedback.Busy 				:= TRUE;
	
	THIS^.fbMoveAbsoluteCA[nInactiveInstance].ContinuousUpdate := TRUE;
	THIS^.fbMoveAbsoluteCA[nInactiveInstance].Execute		:= TRUE;
	THIS^.fbMoveAbsoluteCA[nInactiveInstance].Gap			:= lrGap;
	THIS^.fbMoveAbsoluteCA[nInactiveInstance].Position		:= lrPosition;
	THIS^.fbMoveAbsoluteCA[nInactiveInstance].Direction		:= Direction;
	THIS^.fbMoveAbsoluteCA[nInactiveInstance].BufferMode 	:= BufferMode;
	
	//If the currend command is a buffered movement, then set a flag.
	IF BufferMode <> MC_BufferMode.MC_Aborting THEN
		bNewBufferCommadThisCycle := TRUE;
	END_IF
	
	//Velocity
	//If input = 0  then use default dynamics
	IF lrVelocity = 0.0 THEN
		THIS^.fbMoveAbsoluteCA[nInactiveInstance].Velocity := THIS^.lrDefaultVelocity;
	ELSE
		THIS^.fbMoveAbsoluteCA[nInactiveInstance].Velocity := lrVelocity;
	END_IF
	
	//Acceleration
	//If input = 0  then use default dynamics
	IF lrAcceleration = 0.0 THEN
		THIS^.fbMoveAbsoluteCA[nInactiveInstance].Acceleration := THIS^.lrDefaultAcceleration;
	ELSE
		THIS^.fbMoveAbsoluteCA[nInactiveInstance].Acceleration := lrAcceleration;
	END_IF
	
	//Deceleration
	//If input = 0  then use default dynamics
	IF lrDeceleration = 0.0 THEN
		THIS^.fbMoveAbsoluteCA[nInactiveInstance].Deceleration := THIS^.lrDefaultDeceleration;
	ELSE
		THIS^.fbMoveAbsoluteCA[nInactiveInstance].Deceleration := lrDeceleration;
	END_IF
	
	//Jerk
	//If input = 0  then use default dynamics
	IF lrJerk = 0.0 THEN
		THIS^.fbMoveAbsoluteCA[nInactiveInstance].Jerk := THIS^.lrDefaultJerk;
	ELSE
		THIS^.fbMoveAbsoluteCA[nInactiveInstance].Jerk := lrJerk;
	END_IF

END_IF


MoveAbsoluteCA := THIS^.fbFeedback;
END_METHOD

METHOD Update  : HRESULT
// ********************** Do initialisation first ***********************************************
IF NOT bInitDone THEN
	Update := THIS^.Initialize();
	RETURN;
END_IF

// ********************** Set feedback depending on active command *******************************
CASE THIS^.eActiveCommand OF                                                                      
	E_NcAxisCommands.MoveAbsoluteCA:                                                              
		fbFeedback.Busy 		:= fbMoveAbsoluteCA[nActiveMoveAbsCa].Busy;                       
		fbFeedback.Done 		:= fbMoveAbsoluteCA[nActiveMoveAbsCa].Done;                       
		fbFeedback.ErrorId 		:= fbMoveAbsoluteCA[nActiveMoveAbsCa].ErrorID;  
       
	E_NcAxisCommands.HaltCA:                                                              
		fbFeedback.Busy 		:= fbHaltCA.Busy;                       
		fbFeedback.Done 		:= fbHaltCA.Done OR fbHaltCA.CommandAborted;                       
		fbFeedback.ErrorId 		:= fbHaltCA.ErrorID;            
END_CASE                                                                                          

// **********************  Cyclic call super Update  *********************************************************
SUPER^.Update();
                                                                                                  
                                                                                                  
// **********************  Cyclic calls  *********************************************************
fbMoveAbsoluteCA[0](Axis := THIS^.Axis);                                                          
fbMoveAbsoluteCA[1](Axis := THIS^.Axis);                                                          
fbHaltCA(Axis := THIS^.Axis);
                                                                                                
                                                                                                  
// ********************** Reset all Execution flags **********************************************
fbMoveAbsoluteCA[0].Execute := FALSE;                                                             
fbMoveAbsoluteCA[1].Execute := FALSE;
fbHaltCA.Execute := FALSE;                                                                                                  

                                                                                                 
// ****************Get the acive instance. Stay at the last active.*******************************
IF fbMoveAbsoluteCA[0].Active THEN                                                                
	nActiveMoveAbsCa := 0;
ELSIF fbMoveAbsoluteCA[1].Active THEN
	nActiveMoveAbsCa := 1;
END_IF

//Return
Update := THIS^.fbFeedback.HR;
END_METHOD

END_FUNCTION_BLOCK

// COMPENENTs/Mover/FB_XTS_Mover
{attribute 'no_explicit_call' := 'Do not call the body - Stick to OOP'}
FUNCTION_BLOCK FB_XTS_Mover EXTENDS FB_CH_Object IMPLEMENTS I_XTS_Mover, I_XTS_Mover_PLC
VAR	
	//Link to NC
	Axis : FB_XTS_Axis;
	
	{attribute 'hide'}
	bInitDone : BOOL;
	{attribute 'hide'}
	_bInGroup : BOOL;	
	{attribute 'hide'}
	iXtsSystem : I_XTS_System_Registration;
	{attribute 'hide'}
	iUtilityMover : I_TcIoXtsXpuMover;
	{attribute 'hide'}
	fbActiveCmd : FB_CH_Feedback;
	{attribute 'hide'}
	_iParentStation : I_XTS_Station;	
	{attribute 'hide'}
	_NextMover : I_XTS_Mover;
	{attribute 'hide'}
	_TargedStation : STRING;
	{attribute 'hide'}
	_MoveAbsPosition : LREAL;
	{attribute 'hide'}
	_MoveAbsVelocity : LREAL;
	{attribute 'hide'}	
	_Gap 	: LREAL;
	{attribute 'hide'}	
	lrTrackLentgh 			: LREAL; //[mm]  Modulo
	{attribute 'hide'}
	fbFeedback 					: FB_CH_Feedback;
	
END_VAR
VAR PERSISTENT
	{attribute 'hide'}
	_DrivenDistance : LREAL;
END_VAR

METHOD Disable : HRESULT
Axis.PowerOff();

IF Axis.Feedback.LastCommandAccepted THEN
	Disable := S_OK;
ELSE  
	Disable := E_FAIL;;	
END_IF


//Show as feedback the state of the includet axis
fbFeedback.ActiveCommand := Axis.Feedback.ActiveCommand;
fbFeedback.LastCommandAccepted := Axis.Feedback.LastCommandAccepted;
fbFeedback.HR := Axis.Feedback.hr;
END_METHOD

METHOD Enable : HRESULT
Axis.PowerOn();

IF Axis.Feedback.LastCommandAccepted THEN
	Enable := S_OK;
ELSE  
	Enable := E_FAIL;;	
END_IF


//Show as feedback the state of the includet axis
fbFeedback.ActiveCommand := Axis.Feedback.ActiveCommand;
fbFeedback.LastCommandAccepted := Axis.Feedback.LastCommandAccepted;
fbFeedback.HR := Axis.Feedback.hr;
END_METHOD

METHOD HaltCA : HRESULT
VAR_INPUT
END_VAR
Axis.HaltCA(
	lrDeceleration:= 0, //use default
	lrJerk:= 0, //use default
	lrGap:= _Gap);
	
IF Axis.Feedback.LastCommandAccepted THEN
	HaltCA := S_OK;
ELSE  
	HaltCA := E_FAIL;;	
END_IF


//Show as feedback the state of the includet axis
fbFeedback.ActiveCommand := Axis.Feedback.ActiveCommand;
fbFeedback.LastCommandAccepted := Axis.Feedback.LastCommandAccepted;
fbFeedback.HR := Axis.Feedback.hr;
END_METHOD

METHOD MoveAbsCA : HRESULT
VAR_INPUT
	Position	: LREAL := MC_INVALID;
	Velocity	: LREAL := MC_INVALID;
	Gap			: LREAL := MC_DEFAULT;
	Direction	: Tc3_Mc3Definitions.MC_DIRECTION;
END_VAR
Axis.MoveAbsoluteCA(
	lrPosition:= Position, 
	lrVelocity:= Velocity, 
	lrGap:= Gap, 
	lrAcceleration:= 0, 
	lrDeceleration:= 0, 
	lrJerk:= 0, 
	Direction := Direction,
	BufferMode:= MC_BUFFER_MODE.mcAborting);

THIS^._MoveAbsVelocity := Velocity;
THIS^._MoveAbsPosition := Position;
THIS^._Gap := Gap;

IF Axis.Feedback.LastCommandAccepted THEN
	MoveAbsCA := S_OK;
ELSE  
	MoveAbsCA := E_FAIL;;	
END_IF


//Show as feedback the state of the includet axis
fbFeedback.ActiveCommand := Axis.Feedback.ActiveCommand;
fbFeedback.LastCommandAccepted := Axis.Feedback.LastCommandAccepted;
fbFeedback.HR := Axis.Feedback.hr;
END_METHOD

METHOD Reset : HRESULT
Axis.Reset();

IF Axis.Feedback.LastCommandAccepted THEN
	Reset := S_OK;
ELSE  
	Reset := E_FAIL;;	
END_IF


//Show as feedback the state of the includet axis
fbFeedback.ActiveCommand := Axis.Feedback.ActiveCommand;
fbFeedback.LastCommandAccepted := Axis.Feedback.LastCommandAccepted;
fbFeedback.HR := Axis.Feedback.hr;
END_METHOD

{attribute 'monitoring':='call'}
PROPERTY Coupled : BOOL
GET
Coupled := THIS^.Axis.Coupled;
END_GET
END_PROPERTY

{attribute 'monitoring':='call'}
PROPERTY DrivenDistance : LREAL
GET
DrivenDistance := _DrivenDistance;
END_GET
END_PROPERTY

{attribute 'monitoring':='call'}
PROPERTY Feedback : I_CH_Feedback
GET
Feedback := THIS^.fbFeedback;
END_GET
END_PROPERTY

{attribute 'monitoring':='call'}
PROPERTY Gap : LREAL
GET
Gap := _Gap;
END_GET
END_PROPERTY

PROPERTY getAxisRef : REFERENCE TO Tc2_MC2.AXIS_REF
GET
getAxisRef REF= THIS^.Axis.getAxisRef;
END_GET
END_PROPERTY

PROPERTY IdentInGroup : IDENT_IN_GROUP_REF
GET
IdentInGroup := UDINT_TO_IDENTINGROUP(THIS^.Axis.getAxisRef.NcToPlc.AxisId);
END_GET
END_PROPERTY

{attribute 'monitoring':='call'}
PROPERTY LagDistance : LREAL
GET
LagDistance := THIS^.Axis.LagDistance;
END_GET
END_PROPERTY

{attribute 'monitoring':='call'}
PROPERTY MoveAbsPosition : LREAL
GET
MoveAbsPosition := _MoveAbsPosition;
END_GET
END_PROPERTY

{attribute 'monitoring':='call'}
PROPERTY MoveAbsVelocity : LREAL
GET
MoveAbsVelocity := _MoveAbsVelocity;
END_GET
END_PROPERTY

{attribute 'monitoring':='call'}
PROPERTY MoverInGroup : BOOL
GET
MoverInGroup := _bInGroup;
END_GET
SET
_bInGroup := MoverInGroup;
END_SET
END_PROPERTY

{attribute 'monitoring':='call'}
PROPERTY Moving : BOOL
GET
Moving := THIS^.Axis.Moving;
END_GET
END_PROPERTY

{attribute 'monitoring':='call'}
PROPERTY NextMover : I_XTS_Mover
GET
NextMover := _NextMover;
END_GET
END_PROPERTY

{attribute 'monitoring':='call'}
PROPERTY OID : OTCID
GET
OID := THIS^.Axis.OID;
END_GET
END_PROPERTY

{attribute 'monitoring':='call'}
PROPERTY ParentStation : I_XTS_Station
GET
ParentStation := _iParentStation;
END_GET
SET
_iParentStation := ParentStation;
END_SET
END_PROPERTY

{attribute 'monitoring':='call'}
PROPERTY PositionOnTrack : LREAL
GET
//Round to 3 digits. If Axis is not enabled, use act position
IF THIS^.Axis.getAxisRef.Status.Disabled THEN
	PositionOnTrack := TO_LREAL(TRUNC(THIS^.Axis.ActPosModulo*1000))/1000;
ELSE
	PositionOnTrack := TO_LREAL(TRUNC(THIS^.Axis.SetPosModulo*1000))/1000;	
END_IF
END_GET
END_PROPERTY

{attribute 'monitoring':='call'}
PROPERTY SetAcceleration : LREAL
GET
SetAcceleration := THIS^.Axis.SetAcceleration;
END_GET
END_PROPERTY

{attribute 'monitoring':='call'}
PROPERTY SetVelocity : LREAL
GET
SetVelocity := THIS^.Axis.SetVelocity;
END_GET
END_PROPERTY

{attribute 'monitoring':='call'}
PROPERTY TargedStation : STRING
GET
TargedStation := _TargedStation;
END_GET
SET
_TargedStation := TargedStation;
END_SET
END_PROPERTY

METHOD FB_init : BOOL
VAR_INPUT
	bInitRetains : BOOL; // if TRUE, the retain variables are initialized (warm start / cold start)
	bInCopyCode : BOOL;  // if TRUE, the instance afterwards gets moved into the copy code (online change)
	
	iXtsSystem : I_XTS_System_Registration; //Interface to XTS system object
END_VAR
//Regristrate object in System
IF iXtsSystem <> 0 THEN
	iXtsSystem.RegisterMover(THIS^);
	THIS^.iXtsSystem := iXtsSystem;
END_IF
END_METHOD

METHOD Initialize : HRESULT
VAR
	iTempMover : I_XTS_Mover;
	nLoopIndex : UINT;
END_VAR
fbFeedback.hr := S_OK;	

IF NOT THIS^.bInitDone THEN
	fbFeedback.ActiveCommand := 'Init';
	
	//Get Tracklength from system
	THIS^.lrTrackLentgh := THIS^.iXtsSystem.TrackLength;
	
	
	//Validate Settings
	IF (lrTrackLentgh <= 0) THEN
			fbFeedback.hr := GetMostSignificant(fbFeedback.hr, E_FAIL);		
	END_IF
	

	//If only one mover is in project, then interface stays 0.
	IF THIS^.iXtsSystem.Movers.Size > 1 THEN
		THIS^._NextMover := THIS^.iXtsSystem.getMoverInFront(THIS^);
		//Validate Settings
		IF (_NextMover = 0) THEN
			fbFeedback.hr := GetMostSignificant(fbFeedback.hr, E_FAIL);	
		END_IF
	ELSE
		THIS^._NextMover := 0;
	END_IF
	
	// Get XTS Utility mover object
	IF iXtsSystem.Environment <> 0 THEN
		iUtilityMover := iXtsSystem.Environment.UtilityEnvirement.GetMoverInterfaceByAxisId(THIS^.getAxisRef.NcToPlc.AxisId);
	END_IF
	
	
	//InitAxis
	fbFeedback.hr := GetMostSignificant(fbFeedback.hr, Axis.Initialize());	

	bInitDone := CheckOk(fbFeedback.hr);
END_IF

Initialize := fbFeedback.hr;
END_METHOD

METHOD Update : HRESULT
VAR
	lrDistanceThisCycle : LREAL;
END_VAR
VAR_INST
	lrLastMoverPosition : LREAL;
END_VAR
// Total distance traveled by the mover
IF Axis.Moving THEN
	lrDistanceThisCycle := ABS(Axis.SetPosModulo-lrLastMoverPosition);
	IF lrDistanceThisCycle > (THIS^.lrTrackLentgh*0.5) THEN
		lrDistanceThisCycle := THIS^.lrTrackLentgh-lrDistanceThisCycle;
	END_IF
	_DrivenDistance := _DrivenDistance + lrDistanceThisCycle;
END_IF

lrLastMoverPosition := Axis.SetPosModulo;

Axis.Update();

//Show as feedback the state of the includet axis
fbFeedback.ActiveCommand := Axis.Feedback.ActiveCommand;
fbFeedback.HR := Axis.Feedback.hr;
END_METHOD

{attribute 'monitoring':='call'}
PROPERTY UtilityMover : I_TcIoXtsXpuMover
GET
UtilityMover := iUtilityMover;
END_GET
END_PROPERTY

END_FUNCTION_BLOCK

// COMPENENTs/Station/FB_XTS_Station
{attribute 'no_explicit_call' := 'Do not call the body - Stick to OOP'}
FUNCTION_BLOCK FB_XTS_Station EXTENDS FB_CH_Object IMPLEMENTS I_XTS_Station, I_XTS_Station_PLC
VAR
	{attribute 'hide'}
	bInitDone : BOOL;
	{attribute 'hide'}
	iXtsSystem : I_XTS_System_Registration;
	
	{attribute 'hide'}	
	_StationInFront 			: I_XTS_Station;
	{attribute 'hide'}	
	_StationBehinde 			: I_XTS_Station;
	{attribute 'hide'}
	_StationID 					: STRING;
	{attribute 'hide'}
	_MoverGapAtExit 			: LREAL;
	{attribute 'hide'}
	_MoverVelocityAtExit		: LREAL;	
	{attribute 'hide'}
	_PositionOnTrack 			: LREAL;
	{attribute 'hide'}
	_MoverQueueSize 			: UINT;
	{attribute 'hide'}	
	lrTrackLentgh 				: LREAL; //[mm]  Modulo
	{attribute 'hide'}
	fbAssignedMovers 			: FB_CH_List;		// List of movers approaching the station
	{attribute 'hide'}
	fbFeedback 					: FB_CH_Feedback;
	{attribute 'hide'}
	_SuppressDynamicsChange		: BOOL;
	
	{attribute 'TcInitSymbol'}
	OIDStationInfo : OTCID; //OID of XtsStationInfo object to visualize in Viewer. 0 if not used.
	{attribute 'hide'}
	iStationInfo : I_TcIoXtsInfoServerInfoStation;
	
	// iXtsIsNotValid at this point, call the konstruktor again in the FB_Init
	{attribute 'hide'}
	fbTrigger 					: FB_XTS_Trigger(iXtsSystem);
	{attribute 'hide'}
	fbSortedListMoversInQueue	: FB_XTS_Zone(iXtsSystem);
END_VAR

METHOD AddMoverToQueue : HRESULT
VAR_INPUT
	iMover : I_XTS_Mover;
END_VAR
VAR
	iObject : I_CH_Object;
END_VAR
//Get I_CH_Objekt of mover to put it in to a list.
IF iMover <> 0 AND_THEN __QUERYINTERFACE(iMover,iObject) THEN
	//Add in List of Movers in this station
	THIS^.fbAssignedMovers.AddObject(iObject);
	
	//Handover information in Mover
	iMover.ParentStation := (THIS^);

	AddMoverToQueue := S_OK;
END_IF
END_METHOD

{attribute 'monitoring':='call'}
PROPERTY AreMoversInPlace : BOOL
GET
VAR
	tempMoverInPosition : BOOL;
	nLoopIndex : UINT;
	lrExpectedPosition : LREAL;
END_VAR
//If queuesize is zero, mover is never in place.
IF _MoverQueueSize = 0 THEN
	fbFeedback.HR := E_FAIL;
	RETURN;
END_IF


tempMoverInPosition := TRUE;
lrExpectedPosition := THIS^._PositionOnTrack;
FOR nLoopIndex := 0 TO (THIS^._MoverQueueSize-1) DO
	IF THIS^.fbSortedListMoversInQueue.MoversInZone[nLoopIndex] <> 0 THEN
		
		//Check position and Gap
		IF nLoopIndex <> 0 THEN
			lrExpectedPosition := lrExpectedPosition - THIS^.fbSortedListMoversInQueue.MoversInZone[nLoopIndex].Gap;
			IF lrExpectedPosition < 0 THEN 
				lrExpectedPosition := lrExpectedPosition + lrTrackLentgh;
			END_IF
		END_IF
		tempMoverInPosition := tempMoverInPosition AND (ABS(THIS^.fbSortedListMoversInQueue.MoversInZone[nLoopIndex].PositionOnTrack - lrExpectedPosition) <= 0.05 ); // ToDo: Genauigkeit parametrierbar machen?
		
		//Check if velocity is 0
		tempMoverInPosition := tempMoverInPosition AND (THIS^.fbSortedListMoversInQueue.MoversInZone[nLoopIndex].SetVelocity = 0.0);
		
		//Check mover has this station as targed
		tempMoverInPosition := tempMoverInPosition AND (THIS^.fbSortedListMoversInQueue.MoversInZone[nLoopIndex].TargedStation = THIS^.StationGroupID);
	ELSE	
		tempMoverInPosition := FALSE;
		RETURN;
	END_IF
END_FOR

AreMoversInPlace := tempMoverInPosition;
END_GET
END_PROPERTY

{attribute 'monitoring':='call'}
PROPERTY CtsEmptySpaceInQueue : UINT
GET
//Handle UINT Overflow
IF THIS^.fbAssignedMovers.Size >= THIS^._MoverQueueSize THEN
	CtsEmptySpaceInQueue := 0;
ELSE 
	CtsEmptySpaceInQueue := THIS^._MoverQueueSize - THIS^.fbAssignedMovers.Size;
END_IF
END_GET
END_PROPERTY

{attribute 'monitoring':='call'}
PROPERTY CtsMoversInQueue : UINT
GET
CtsMoversInQueue := THIS^.fbAssignedMovers.Size;
END_GET
END_PROPERTY

METHOD DeleteMoversQueue : HRESULT
THIS^.fbAssignedMovers.Clear();
DeleteMoversQueue := S_OK;
END_METHOD

METHOD FB_init : BOOL
VAR_INPUT
	bInitRetains : BOOL; // if TRUE, the retain variables are initialized (warm start / cold start)
	bInCopyCode : BOOL;  // if TRUE, the instance afterwards gets moved into the copy code (online change)
	
	iXtsSystem : I_XTS_System_Registration; //Interface to XTS system object
	PositionOnTrack 		: LREAL;	//[mm]
	StationID 				: STRING;	//expl.:'Loading'
	MoverQueueSize 			: UINT;		//[cts]
	
	//Dynamik at exit of station
	MoverGapAtExit 			: LREAL;	//[mm]
	MoverVelocityAtExit 	: LREAL;	//[mm/s]

END_VAR
//Regristrate object in System
IF iXtsSystem <> 0 THEN
	iXtsSystem.RegisterStation(THIS^);
	THIS^.iXtsSystem := iXtsSystem;
END_IF

THIS^._StationID := StationID;
THIS^._MoverGapAtExit := MoverGapAtExit;
THIS^._MoverVelocityAtExit := MoverVelocityAtExit;
THIS^._MoverQueueSize := MoverQueueSize;
THIS^._PositionOnTrack := PositionOnTrack;

THIS^.fbTrigger.FB_init(FALSE,FALSE, iXtsSystem);
THIS^.fbSortedListMoversInQueue.FB_init(FALSE,FALSE, iXtsSystem);
END_METHOD

{attribute 'monitoring':='call'}
PROPERTY HR : HRESULT
GET
HR := fbFeedback.hr;
END_GET
END_PROPERTY

METHOD Initialize : HRESULT
VAR
	nLoopIndex : UINT;
	iTempStation : I_XTS_Station;
	
	//Utility InfoStation, used in XTS Viewer
	aStopPositionsInfoStation : ARRAY[1..Tc3_XTS_Utility.TcIoXtsEnvironmentParameterList.MaxXtsStopPositionsPerStation] OF LREAL;
	fLastStopPosition : LREAL;
	
    iMovers : CHALET_BaseComponents.I_CH_List;
	iTempMover : I_XTS_Mover;
	anBias : ARRAY[1..2] OF INT;
	bInverted : BOOL;
END_VAR
fbFeedback.hr := S_OK;	

IF NOT THIS^.bInitDone THEN
	THIS^.lrTrackLentgh := THIS^.iXtsSystem.TrackLength;
	THIS^._StationInFront := THIS^.iXtsSystem.getStationInFront(THIS^);
	
	//Init Tigger
	fbFeedback.hr := GetMostSignificant(S_OK,fbTrigger.Initialize());	
	
	fbTrigger.ListOfMoversToCheck := THIS^.iXtsSystem.Movers;
	fbTrigger.PositionOnTrack := THIS^.PositionOnTrack;
	fbTrigger.TriggerDirection := MC_Positive_Direction;
	
	//Use the zone to sort all movers in this queue depending on the distance to targed in an output array.
	//The Zone is set to the length of the whole system, but only add the mover in the station queue.
	fbFeedback.hr := GetMostSignificant(fbFeedback.hr,fbSortedListMoversInQueue.Initialize());		
	fbSortedListMoversInQueue.EndPositionOnTrack := THIS^.PositionOnTrack;
	fbSortedListMoversInQueue.StartPositionOnTrack := (THIS^.PositionOnTrack + 0.1);
	fbSortedListMoversInQueue.ListOfMoversToCheck := THIS^.fbAssignedMovers;
	
	
	//Get Station behinde this one.
	iTempStation := (THIS^);
	WHILE((iTempStation <> 0) AND_THEN (iTempStation.StationInFront <> 0)) DO
		// test if this is the station behinde
		IF (iTempStation.StationInFront.StationGroupID = THIS^.StationGroupID) THEN
			THIS^._StationBehinde := iTempStation;	
			EXIT;	
		END_IF
		// get Next Stations
		iTempStation := iTempStation.StationInFront;
	END_WHILE


	
	//Validate Settings - Pending
	IF (_StationBehinde = 0) THEN
			fbFeedback.hr := GetMostSignificant(S_Pending, fbFeedback.hr);
	END_IF
	
	
	//Validate Settings - Error
	IF ((_StationInFront = 0) AND (_StationID = '') AND (lrTrackLentgh <= 0) AND (_PositionOnTrack < 0.0) AND (_PositionOnTrack >= lrTrackLentgh) AND (_MoverVelocityAtExit <= 0) AND (_MoverGapAtExit <= 0)) THEN
			fbFeedback.hr := GetMostSignificant(E_FAIL, fbFeedback.hr);
	END_IF

	
	// callculate Position Offset
	iMovers := iXtsSystem.Movers;
	iMovers.ResetIterator();
	nLoopIndex := 0;	
	WHILE iMovers.HasNextObject() DO
		nLoopIndex := nLoopIndex + 1;
		IF ToMover(iMovers.GetNextObject(),iTempMover) THEN
			anBias[nLoopIndex] := LREAL_TO_INT(iXtsSystem.Environment.UtilityEnvirement.XpuTcIo(1).MoverTcIo(nLoopIndex).GetPositionInfo().fPartPosition - iTempMover.getAxisRef.NcToPlc.ModuloActPos);
			IF nLoopIndex = 2 THEN
				 EXIT;
			END_IF
		END_IF
	END_WHILE
	
	// validate bias, check for inverted direction
	IF anBias[1] <> anBias[2] THEN
		bInverted := TRUE; 
		iMovers.ResetIterator();
		nLoopIndex := 0;	
		WHILE iMovers.HasNextObject() DO
			nLoopIndex := nLoopIndex + 1;
			IF ToMover(iMovers.GetNextObject(),iTempMover) THEN
				anBias[nLoopIndex] := LREAL_TO_INT(iXtsSystem.TrackLength - iXtsSystem.Environment.UtilityEnvirement.XpuTcIo(1).MoverTcIo(nLoopIndex).GetPositionInfo().fPartPosition - iTempMover.getAxisRef.NcToPlc.ModuloActPos);
				IF nLoopIndex = 2 THEN
					 EXIT;
				END_IF
			END_IF	
		END_WHILE
	END_IF
	
	//Utility InfoStation, used in XTS Viewer
	IF THIS^.OIDStationInfo <> 0 AND iXtsSystem.Environment <> 0 THEN
		//Get interface to utility station belongs to this station via OID
		FOR nLoopIndex := 1 TO iXtsSystem.Environment.UtilityEnvirement.InfoServerTcIo(1).P_InfoStationCount DO
			IF 	iXtsSystem.Environment.UtilityEnvirement.InfoServerTcIo(1).P_InfoStationOids[nLoopIndex] = THIS^.OIDStationInfo THEN
				THIS^.iStationInfo := iXtsSystem.Environment.UtilityEnvirement.InfoServerTcIo(1).InfoStationTcIo(nInfoStation:= nLoopIndex);
				EXIT;
			END_IF
		END_FOR

		//configure/draw station in viewer
		IF THIS^.iStationInfo <> 0 THEN		
			// draw stop position if gap between mover, given by station behind, is set
			IF (StationBehinde <> 0) AND (THIS^._MoverQueueSize > 0) AND THIS^._MoverQueueSize <= 25 THEN
				//Clear array
				MEMSET(ADR(aStopPositionsInfoStation), SIZEOF(aStopPositionsInfoStation), 0);
				//Fill array
				FOR nLoopIndex := 1 TO THIS^._MoverQueueSize DO
					fLastStopPosition := (nLoopIndex-1)*StationBehinde.MoverGapAtExit;
					aStopPositionsInfoStation[(nLoopIndex)] := (fLastStopPosition);
				END_FOR
				IF NOT bInverted THEN
					//Start Position
					THIS^.iStationInfo.SetStartPositionOnPart(MAX((_PositionOnTrack + anBias[1] - fLastStopPosition), 0)); ///zzz Todo. The InfoStation can not draw stations in the modulo area
					//End Pos
					THIS^.iStationInfo.SetEndPositionOnPart(_PositionOnTrack + anBias[1]);
				ELSE
					//Start Position
					THIS^.iStationInfo.SetStartPositionOnPart(iXtsSystem.TrackLength - (_PositionOnTrack + anBias[1]));					
					//End Pos
					THIS^.iStationInfo.SetEndPositionOnPart(MAX((iXtsSystem.TrackLength - (_PositionOnTrack + anBias[1] - fLastStopPosition)), 0)); ///zzz Todo. The InfoStation can not draw stations in the modulo area
				END_IF
				//StopPositions
				THIS^.iStationInfo.SetStopPositions(aStopPositionsInfoStation);

				//Override color if is set to transparent
				IF THIS^.iStationInfo.GetStationColor() = 0 THEN
					THIS^.iStationInfo.SetStationColor(nStationColor:= E_Colors_ARGB.Darkred);
				END_IF
			ELSE
				//Clear array
				MEMSET(ADR(aStopPositionsInfoStation), SIZEOF(aStopPositionsInfoStation), 0);	
				//StopPositions
				THIS^.iStationInfo.SetStopPositions(aStopPositionsInfoStation);
				//Start Pos
				THIS^.iStationInfo.SetStartPositionOnPart(nStartPositionOnPart := _PositionOnTrack + anBias[1]);
				//End Position
				THIS^.iStationInfo.SetEndPositionOnPart(nEndPositionOnPart := _PositionOnTrack + anBias[1]);
			END_IF
		END_IF
	END_IF
	
	
	bInitDone := CheckOk(fbFeedback.hr);
END_IF

				
								
Initialize := fbFeedback.hr;
END_METHOD

{attribute 'monitoring':='call'}
PROPERTY LUID : STRING
GET
LUID := _StationID;
END_GET
END_PROPERTY

{attribute 'monitoring':='call'}
PROPERTY MoverGapAtExit : LREAL //[mm]
GET
MoverGapAtExit := _MoverGapAtExit;
END_GET
SET
_MoverGapAtExit := MoverGapAtExit;
END_SET
END_PROPERTY

{attribute 'monitoring':='call'}
PROPERTY MoverQueueSize : UINT
GET
MoverQueueSize := THIS^._MoverQueueSize;
END_GET
SET
THIS^._MoverQueueSize := MoverQueueSize;
END_SET
END_PROPERTY

{attribute 'monitoring':='call'}
PROPERTY MoversInQueue : REFERENCE TO ARRAY [0..(XtsParameterlist.MAX_MOVER_PER_SYSTEM-1)] OF I_XTS_Mover_PLC // Return a sorted list of movers in this zone. Index 0 is the mover in Front.
GET
MoversInQueue REF= THIS^.fbSortedListMoversInQueue.MoversInZone;
END_GET
END_PROPERTY

{attribute 'monitoring':='call'}
PROPERTY MoverVelocityAtExit : LREAL //[mm/s]
GET
MoverVelocityAtExit := _MoverVelocityAtExit;
END_GET
SET
_MoverVelocityAtExit := MoverVelocityAtExit;
END_SET
END_PROPERTY

{attribute 'monitoring':='call'}
PROPERTY OID : OTCID
GET
OID := THIS^.OIDStationInfo;
END_GET
END_PROPERTY

{attribute 'monitoring':='call'}
PROPERTY PositionOnTrack : LREAL
GET
PositionOnTrack := _PositionOnTrack;
END_GET
END_PROPERTY

METHOD SendMoversToStation : HRESULT //Send the 
VAR_INPUT
	TargedStation	: STRING;
END_VAR
VAR
	nLoopIndex 		: UINT;;
	iMover	: I_XTS_Mover;
END_VAR
//Invalide targed
IF TargedStation = '' THEN
	SendMoversToStation := E_FAIL;
	RETURN;
END_IF

//Movers have not reached station and can not send away until complet
IF NOT THIS^.AreMoversInPlace THEN
	SendMoversToStation := E_FAIL;
	RETURN;
END_IF

//Send all Queued movers away by changing the targed station destination
FOR nLoopIndex := 0 TO _MoverQueueSize-1 DO
	IF THIS^.MoversInQueue[nLoopIndex] <> 0 AND_THEN __QUERYINTERFACE(THIS^.MoversInQueue[nLoopIndex],iMover) THEN
		iMover.TargedStation := TargedStation;		
	END_IF
END_FOR
END_METHOD

{attribute 'monitoring':='call'}
PROPERTY StationBehinde : I_XTS_Station
GET
StationBehinde := _StationBehinde;
END_GET
END_PROPERTY

{attribute 'monitoring':='call'}
PROPERTY StationGroupID : STRING
GET
StationGroupID := _StationID;
END_GET
END_PROPERTY

{attribute 'monitoring':='call'}
PROPERTY StationInFront : I_XTS_Station
GET
StationInFront := _StationInFront;
END_GET
END_PROPERTY

{attribute 'monitoring':='call'}
PROPERTY SuppressDynamicsChange : BOOL
GET
SuppressDynamicsChange := _SuppressDynamicsChange;
END_GET
SET
_SuppressDynamicsChange := SuppressDynamicsChange;
END_SET
END_PROPERTY

//This sequence tries to transfer the mover to the next station in the direction of travel and checks whether the next station has space for it. 
//If the next station is a "dummy" that only changes the dynamics of the passing mover, this station is skipped and the next station is searched one ahead.
//If the station is fully occupied, no action is taken and a new search can be made in the next cycle.
METHOD PRIVATE TrySendMoverToNextStation : HRESULT
VAR_INPUT
	iMover	: I_XTS_Mover;
	Velocity : LREAL;
	Gap : LREAL;
END_VAR
VAR
	bStationIsOnlyForDynamicChanges : BOOL;
	bStationIsFull					: BOOL;
	bStationHanMoreMoverThanAllowed : BOOL;
	bStationHasAFreePlaceInQueue 	: BOOL;
	bStationIsTheTarged				: BOOL;
	
	iMoverObject 		: I_CH_Object;
	iTempStation 	: I_XTS_Station;	
	iTargedStation 	: I_XTS_Station;

	stCommand : ST_TcIoXtsMoverCommand;	
END_VAR
//Invalide interface
IF iMover = 0 THEN
	TrySendMoverToNextStation := E_FAIL;
	RETURN;
END_IF

//Mover is not in this Station.
IF __QUERYINTERFACE(iMover,iMoverObject) AND_THEN NOT THIS^.fbAssignedMovers.FindObject(iMoverObject) THEN
	TrySendMoverToNextStation := E_FAIL;
	RETURN;
END_IF

//Send to actual Station is not supported
IF iMover.TargedStation = THIS^.StationGroupID THEN
	TrySendMoverToNextStation := E_FAIL;
	RETURN;
END_IF


iTempStation := (THIS^);
//This sequence tries to transfer the mover to the next station in the direction of travel and checks whether the next station has space for it. 
//If the next station is a "dummy" that only changes the dynamics of the passing mover, this station is skipped and the next station is searched one ahead.
//If the station is fully occupied, no action is taken and a new search can be made in the next cycle.
WHILE (iTargedStation=0) DO
	
	//get next station in flow direction
	iTempStation := iTempStation.StationInFront;

	//All Stations around the XTS tested, Station not Found
	IF iTempStation.StationGroupID = THIS^.StationGroupID THEN
		TrySendMoverToNextStation := E_FAIL;
		RETURN;
	END_IF

	bStationHanMoreMoverThanAllowed := (iTempStation.CtsMoversInQueue > iTempStation.MoverQueueSize); //Maybe during statup if all movers are forced to station x.	
	bStationIsFull					:= (iTempStation.CtsEmptySpaceInQueue = 0) AND NOT (iTempStation.MoverQueueSize = 0);
	bStationHasAFreePlaceInQueue 	:= (iTempStation.CtsEmptySpaceInQueue > 0);
	bStationIsOnlyForDynamicChanges := (iTempStation.MoverQueueSize = 0);
	bStationIsTheTarged				:= (iTempStation.StationGroupID = iMover.TargedStation);
	
	IF bStationIsFull OR bStationHanMoreMoverThanAllowed THEN
		//Next Station is a valide targed but is already full.  Exit WHILE loop and try again next time.
		EXIT;
	
	ELSIF bStationHasAFreePlaceInQueue THEN
		//Next station found. Send mover to it.
		iTargedStation := iTempStation;
	
	ELSIF bStationIsOnlyForDynamicChanges AND bStationIsTheTarged THEN
		//ERROR. The target position is a dynamic station and can not be reached.
		TrySendMoverToNextStation := E_FAIL;
		RETURN;
		
	ELSIF bStationIsOnlyForDynamicChanges THEN
		//Repead WHILE loop and search an station more in front.
		;
	END_IF 

END_WHILE


//Requested station was found, send movers to there if it has space.
IF iTargedStation <> 0 THEN
	//Handover Mover
	THIS^.fbAssignedMovers.RemoveObject(iMoverObject);
	iTargedStation.AddMoverToQueue(iMover);
	//Start Movement
	iMover.MoveAbsCA(
		Position:= iTargedStation.PositionOnTrack, 
		Velocity:= Velocity, 
		Gap:= Gap, 
		Direction:= Tc3_Mc3Definitions.MC_DIRECTION.mcDirectionPositive);
		
	//Log Command
	stCommand.sCommandType	:= 'leaving station';
	stCommand.sStation		:= iTargedStation.StationGroupID;
	stCommand.sText 		:= FUN_BuildLogString(Pos := iTargedStation.PositionOnTrack, Velocity := Velocity, Gap := Gap);
	iXtsSystem.Environment.UtilityEnvirement.XpuTcIo(1).MoverTcIo(UDINT_TO_UINT(iMover.getAxisRef.NcToPlc.AxisId)).AddCommand(stCommand);
	
	TrySendMoverToNextStation := S_OK;	
ELSE
	//No movemnt possible, try next cycle again		
	TrySendMoverToNextStation := S_FALSE;
END_IF
END_METHOD

METHOD Update : HRESULT
VAR
	iMover : I_XTS_Mover;
END_VAR
//Force to do an init befor call update
IF NOT bInitDone THEN
	THIS^.Initialize();
	RETURN;
END_IF

// If enabled start station logic
IF THIS^.iXtsSystem.Enabled THEN
	
	//Detect mover who is passing the station whitout be in queue. Adjust to new Gap+Dynamics
	IF fbTrigger.MoverDetected AND fbTrigger.MoverAtTrigger<>0 AND NOT THIS^._SuppressDynamicsChange THEN
		fbTrigger.MoverAtTrigger.MoveAbsCA(
			Position:= fbTrigger.MoverAtTrigger.MoveAbsPosition, 
			Velocity:= THIS^._MoverVelocityAtExit, 
			Gap:= THIS^._MoverGapAtExit, 
			Direction:= Tc3_Mc3Definitions.MC_DIRECTION.mcDirectionPositive);
	END_IF
	
	
	//Test if the first mover is in station and send him away, if the destination is not this station
	IF (THIS^.MoversInQueue[0] <> 0) AND_THEN (THIS^.MoversInQueue[0].TargedStation <> THIS^.StationGroupID) AND_THEN __QUERYINTERFACE(THIS^.MoversInQueue[0],iMover) THEN
		//IF mover is standstill in current station, send him away whit the exitVelocity, else use the in mover stored velocity
		IF (THIS^.MoversInQueue[0].PositionOnTrack = THIS^.PositionOnTrack) THEN
			THIS^.TrySendMoverToNextStation(iMover := iMover, Velocity := THIS^._MoverVelocityAtExit, Gap := THIS^._MoverGapAtExit);
		ELSE
			THIS^.TrySendMoverToNextStation(iMover := iMover, Velocity := iMover.MoveAbsVelocity, Gap := iMover.Gap);
		END_IF	
      
	END_IF
END_IF
END_METHOD

PROPERTY UtilityStationInfo : I_TcIoXtsInfoServerInfoStation
GET
UtilityStationInfo := THIS^.iStationInfo;
END_GET
END_PROPERTY

END_FUNCTION_BLOCK

// COMPENENTs/Trigger/FB_XTS_Trigger
{attribute 'no_explicit_call' := 'Do not call the body - Stick to OOP'}
FUNCTION_BLOCK FB_XTS_Trigger EXTENDS FB_CH_Object IMPLEMENTS I_XTS_Trigger
VAR
	{attribute 'hide'}
	bInitDone : BOOL;
	{attribute 'hide'}
	iXtsSystem : I_XTS_System_Registration;
	{attribute 'hide'}
	_iListOfMoversToCheck : I_CH_LIST;
	{attribute 'hide'}
	_PositionOnTrack : LREAL;
	{attribute 'hide'}
	_TriggerDirection : Tc2_MC2.MC_Direction := MC_Positive_Direction;
	{attribute 'hide'}
	_MoverAtTrigger : I_XTS_Mover;
	{attribute 'hide'}	
	lrTrackLentgh : LREAL;
	//{attribute 'hide'}
	aMoversLastPosition : ARRAY [0..(XtsParameterlist.MAX_MOVER_PER_SYSTEM-1)] OF LREAL;
	//{attribute 'hide'}
	aMoversLastMover : ARRAY [0..(XtsParameterlist.MAX_MOVER_PER_SYSTEM-1)] OF I_XTS_Mover;
	
END_VAR

METHOD FB_init : BOOL
VAR_INPUT
	bInitRetains : BOOL; // if TRUE, the retain variables are initialized (warm start / cold start)
	bInCopyCode : BOOL;  // if TRUE, the instance afterwards gets moved into the copy code (online change)
	
	iXtsSystem : I_XTS_System_Registration; //Interface to XTS system object
	
END_VAR
//Regristrate object in System
IF iXtsSystem <> 0 THEN
	iXtsSystem.RegisterTrigger(THIS^);
	THIS^.iXtsSystem := iXtsSystem;
END_IF
END_METHOD

{attribute 'monitoring':='call'}
PROPERTY HR : HRESULT
GET
///zzz todo
END_GET
END_PROPERTY

METHOD Initialize : HRESULT
THIS^.lrTrackLentgh := THIS^.iXtsSystem.TrackLength;

IF (THIS^._iListOfMoversToCheck <> 0) AND (THIS^.lrTrackLentgh > 0.0) THEN
	THIS^.bInitDone := TRUE;
	Initialize := S_OK;
ELSE
	Initialize := E_FAIL;
END_IF
END_METHOD

PROPERTY ListOfMoversToCheck : I_CH_List
SET
IF ListOfMoversToCheck <> 0 THEN
	_iListOfMoversToCheck := ListOfMoversToCheck;
END_IF
END_SET
END_PROPERTY

{attribute 'monitoring':='call'}
PROPERTY MoverAtTrigger : I_XTS_Mover
GET
THIS^.Prepare();//Prepare Time-critical information

MoverAtTrigger := _MoverAtTrigger;
END_GET
END_PROPERTY

{attribute 'monitoring':='call'}
PROPERTY MoverDetected : BOOL
GET
THIS^.Prepare();//Prepare Time-critical information

MoverDetected := (_MoverAtTrigger <> 0);
END_GET
END_PROPERTY

{attribute 'monitoring':='call'}
PROPERTY PositionOnTrack : LREAL
GET
PositionOnTrack := _PositionOnTrack;
END_GET
SET
_PositionOnTrack := PositionOnTrack;
END_SET
END_PROPERTY

(* Time-critical information is processed here, which can then be polled via the property every cycle. 
The update method is usually at the end of the program and then it is already 'outdated'. *)
METHOD PRIVATE Prepare : HRESULT
VAR
	lrActPos,lrLastPos : LREAL;
	lrRangePositive, lrRangeNegative : LREAL;
	bMoverWasInRangeNeg, bMoverWasInRangePos, bMoverIsInRangeNeg, bMoverIsInRangePos : BOOL;
	nLoopIndex : UINT;
END_VAR
VAR_INST
	{attribute 'hide'}
	nLastUpdatedCycleCount : UDINT;
END_VAR
VAR CONSTANT
	lrMaxMoveDistPerCycle : LREAL := 4000.0 * 20.0 / 1000.0 * 1.1; //4 m/s(max. XTS speed) * 20ms(max realistic SPS cycle time) + 10%
END_VAR
//Check if this Cycle the dates are allready prepared
IF nLastUpdatedCycleCount <> TwinCAT_SystemInfoVarList._TaskInfo[THIS^.nTaskIndex].CycleCount THEN
	nLastUpdatedCycleCount := TwinCAT_SystemInfoVarList._TaskInfo[THIS^.nTaskIndex].CycleCount;

	//Clear last stored Mover if an new cycle has started
	THIS^._MoverAtTrigger := 0;
	
	//Check old list of Moverspositions and compare them to the current position of the same mover.
	//Set Trigger if the Mover pass the Station
	lrRangePositive := LMOD(lr_Value:=(THIS^.PositionOnTrack + lrMaxMoveDistPerCycle + THIS^.lrTrackLentgh),lr_Arg:= THIS^.lrTrackLentgh);
	lrRangeNegative := LMOD(lr_Value:=(THIS^.PositionOnTrack - lrMaxMoveDistPerCycle + THIS^.lrTrackLentgh),lr_Arg:= THIS^.lrTrackLentgh);
	
	FOR nLoopIndex := 0 TO (XtsParameterlist.MAX_MOVER_PER_SYSTEM-1) DO
		IF aMoversLastMover[nLoopIndex] <> 0 THEN
			lrActPos :=  aMoversLastMover[nLoopIndex].PositionOnTrack;
			lrLastPos:=  aMoversLastPosition[nLoopIndex];
			
			
			//Test if the the Mover was in Trigger-100mm Range(without exact the trigger point) and is now in Trigger+100 Range(with exact the trigger point)
			bMoverWasInRangePos	:= FUN_InLimitTest(Minimum :=THIS^.PositionOnTrack, Input:= lrLastPos, Maximum:=lrRangePositive) AND NOT (lrLastPos=THIS^.PositionOnTrack); 
			bMoverWasInRangeNeg	:= FUN_InLimitTest(Minimum :=lrRangeNegative, Input:= lrLastPos, Maximum:=THIS^.PositionOnTrack) AND NOT (lrLastPos=THIS^.PositionOnTrack); 
			bMoverIsInRangePos 	:= FUN_InLimitTest(Minimum :=THIS^.PositionOnTrack, Input:= lrActPos, Maximum:=lrRangePositive); 
			bMoverIsInRangeNeg 	:= FUN_InLimitTest(Minimum :=lrRangeNegative, Input:= lrActPos, Maximum:=THIS^.PositionOnTrack); 
		
			IF _TriggerDirection = MC_Positive_Direction AND bMoverWasInRangeNeg AND bMoverIsInRangePos THEN
				THIS^._MoverAtTrigger := aMoversLastMover[nLoopIndex];
				RETURN;
			ELSIF _TriggerDirection = MC_Negative_Direction AND bMoverIsInRangeNeg AND bMoverWasInRangePos THEN
				THIS^._MoverAtTrigger := aMoversLastMover[nLoopIndex];
				RETURN;	
			END_IF
			
		END_IF
	END_FOR
END_IF
END_METHOD

{attribute 'monitoring':='call'}
PROPERTY TimeStamp : Tc2_EtherCAT.T_DCTIME64
GET
THIS^.Prepare();//Prepare Time-critical information

///zzz todo later
 IF _MoverAtTrigger <> 0 THEN
	 TimeStamp := F_GetCurDcTaskTime64();
 ELSE
	 TimeStamp := 0;
 END_IF
END_GET
END_PROPERTY

{attribute 'monitoring':='call'}
PROPERTY TriggerDirection : Tc2_MC2.MC_Direction
GET
TriggerDirection := _TriggerDirection;
END_GET
SET
IF TriggerDirection = MC_Positive_Direction OR TriggerDirection = MC_Negative_Direction THEN
	_TriggerDirection := TriggerDirection;
END_IF
END_SET
END_PROPERTY

METHOD Update : HRESULT
VAR
	nIndex : UINT;
	iMover : I_XTS_Mover;
END_VAR
//Force to do an init befor call update
IF NOT bInitDone THEN
	THIS^.Initialize();
	RETURN;
END_IF

//Clear array
MEMSET(destAddr:=ADR(aMoversLastMover),n:=SIZEOF(aMoversLastMover),fillByte:=0);
MEMSET(destAddr:=ADR(aMoversLastPosition),n:=SIZEOF(aMoversLastPosition),fillByte:=0);

nIndex := 0;
THIS^._iListOfMoversToCheck.ResetIterator();
WHILE THIS^._iListOfMoversToCheck.HasNextObject() DO
	
	//Cheack all Movers fill the actposition in the array
	IF ToMover(THIS^._iListOfMoversToCheck.GetNextObject(),iMover) THEN
		aMoversLastMover[nIndex] := iMover;
		aMoversLastPosition[nIndex] := iMover.PositionOnTrack;
		nIndex := nIndex +1;
	END_IF
	
END_WHILE
END_METHOD

END_FUNCTION_BLOCK

// FUNCTIONs/FUN_InLimitTest
FUNCTION FUN_InLimitTest : BOOL
VAR_INPUT
	Minimum : LREAL;
	Maximum : LREAL;
	Input : LREAL;
END_VAR

//Normal case
// 9 Max
// 5 Test
// 1 Min
IF Minimum <= Maximum THEN
	FUN_InLimitTest := (Input >= Minimum) AND (Input <= Maximum);
	
//Modulo case	
// 6 | 6  Max
// 5 | 9  Test
// 8 | 8  Min
ELSIF Minimum > Maximum THEN
	FUN_InLimitTest := NOT((Input > Maximum) AND (Input < Minimum));
END_IF

END_FUNCTION

// COMPENENTs/Zone/FB_XTS_Zone
{attribute 'no_explicit_call' := 'Do not call the body - Stick to OOP'}
// Check zone start to end in positive direktion.
FUNCTION_BLOCK FB_XTS_Zone EXTENDS FB_CH_Object IMPLEMENTS I_XTS_Zone
VAR
	{attribute 'hide'}
	bInitDone : BOOL;
	{attribute 'hide'}
	iXtsSystem : I_XTS_System_Registration;
	
	//{attribute 'hide'}
	iListOfMoversToCheck : I_CH_LIST;
	//{attribute 'hide'}
	aMoversInZone : ARRAY [0..(XtsParameterlist.MAX_MOVER_PER_SYSTEM-1)] OF I_XTS_Mover_PLC;
	{attribute 'hide'}
	_StartPositionOnTrack : LREAL;
	{attribute 'hide'}
	_EndPositionOnTrack : LREAL;	
	{attribute 'hide'}
	lrTrackLentgh : LREAL;
END_VAR

{attribute 'monitoring':='call'}
PROPERTY CtsMoversInZone : UINT
GET
VAR
	nIndex : UINT;
END_VAR
THIS^.Prepare();//Prepare Time-critical information

//Check array for entrys, exit if fisrt empty arrayindex is found.
FOR nIndex := 0 TO (XtsParameterlist.MAX_MOVER_PER_SYSTEM-1) DO
	IF (aMoversInZone[nIndex] <> 0) THEN
		CtsMoversInZone := CtsMoversInZone +1;
	ELSE
		RETURN;
	END_IF
END_FOR
END_GET
END_PROPERTY

{attribute 'monitoring':='call'}
PROPERTY EndPositionOnTrack : LREAL
GET
EndPositionOnTrack := _EndPositionOnTrack;
END_GET
SET
_EndPositionOnTrack := EndPositionOnTrack;
END_SET
END_PROPERTY

METHOD FB_init : BOOL
VAR_INPUT
	bInitRetains : BOOL; // if TRUE, the retain variables are initialized (warm start / cold start)
	bInCopyCode : BOOL;  // if TRUE, the instance afterwards gets moved into the copy code (online change)
	
	iXtsSystem : I_XTS_System_Registration; //Interface to XTS system object
END_VAR
//Regristrate object in System
IF iXtsSystem <> 0 THEN
	iXtsSystem.RegisterZone(THIS^);
	THIS^.iXtsSystem := iXtsSystem;
END_IF
END_METHOD

{attribute 'monitoring':='call'}
PROPERTY HR : HRESULT
GET
IF CHALET_BaseComponents.BaseParameterlist.MAX_OBJECTS > XtsParameterlist.MAX_MOVER_PER_SYSTEM THEN
	HR := E_FAIL;
END_IF
END_GET
END_PROPERTY

METHOD Initialize : HRESULT
THIS^.lrTrackLentgh := THIS^.iXtsSystem.TrackLength;

IF (THIS^.iListOfMoversToCheck <> 0) AND (THIS^.lrTrackLentgh > 0.0) THEN
	THIS^.bInitDone := TRUE;
	Initialize := S_OK;
ELSE
	Initialize := E_FAIL;
END_IF
END_METHOD

PROPERTY ListOfMoversToCheck : I_CH_List
SET
IF ListOfMoversToCheck <> 0 THEN
	iListOfMoversToCheck := ListOfMoversToCheck;
END_IF
END_SET
END_PROPERTY

{attribute 'monitoring':='call'}
PROPERTY MoversInZone : REFERENCE TO ARRAY [0..(XtsParameterlist.MAX_MOVER_PER_SYSTEM-1)] OF I_XTS_Mover_PLC // Return a sorted list of movers in this zone. Index 0 is the mover in Front.
GET
THIS^.Prepare();//Prepare Time-critical information

MoversInZone REF= THIS^.aMoversInZone;
END_GET
END_PROPERTY

(* Time-critical information is processed here, which can then be polled via the property every cycle. 
The update method is usually at the end of the program and then it is already 'outdated'. *)
METHOD PRIVATE Prepare : HRESULT
VAR
	nLoopIndex : UINT;
	iMoverPlc : I_XTS_Mover_PLC;
	lrDistToStart : LREAL;
	aDisanceToStart : ARRAY [0..XtsParameterlist.MAX_MOVER_PER_SYSTEM] OF LREAL;
END_VAR
VAR_INST
	{attribute 'hide'}
	nLastUpdatedCycleCount : UDINT;
END_VAR
//Check if this Cycle the dates are allready prepared
IF nLastUpdatedCycleCount <> TwinCAT_SystemInfoVarList._TaskInfo[THIS^.nTaskIndex].CycleCount THEN
	nLastUpdatedCycleCount := TwinCAT_SystemInfoVarList._TaskInfo[THIS^.nTaskIndex].CycleCount;

	//Clear array
	MEMSET(destAddr:=ADR(aMoversInZone),n:=SIZEOF(aMoversInZone),fillByte:=0);
	
	//Cheack all Movers and generate a sorted list of all mover in this zone
	THIS^.iListOfMoversToCheck.ResetIterator();
	WHILE THIS^.iListOfMoversToCheck.HasNextObject() DO
		IF ToMover_PLC(THIS^.iListOfMoversToCheck.GetNextObject(),iMoverPlc) THEN
			
			//If in zone
			IF FUN_InLimitTest(Minimum:= _StartPositionOnTrack, Maximum:=_EndPositionOnTrack, Input:= iMoverPlc.PositionOnTrack) THEN
				lrDistToStart := FUN_GetDistToPosModulo(ActualPosition:= iMoverPlc.PositionOnTrack, TargedPosition:= _EndPositionOnTrack, Modulo := lrTrackLentgh);
				
				//Check array of movers and decide if the current one is closer to 
				FOR nLoopIndex := 0 TO (XtsParameterlist.MAX_MOVER_PER_SYSTEM-1) DO
					//empty array position
					IF aMoversInZone[nLoopIndex] = 0 THEN
						aMoversInZone[nLoopIndex] := iMoverPlc;
						aDisanceToStart[nLoopIndex] := lrDistToStart;
						EXIT;
						
					//Closer Mover found, move whole array 	
					ELSIF aDisanceToStart[nLoopIndex] > lrDistToStart THEN
						MEMMOVE(srcAddr := ADR(aMoversInZone[nLoopIndex]), destAddr := ADR(aMoversInZone[nLoopIndex+1]), n := (SIZEOF(aMoversInZone[0])*(XtsParameterlist.MAX_MOVER_PER_SYSTEM-nLoopIndex-1)));
						MEMMOVE(srcAddr := ADR(aDisanceToStart[nLoopIndex]), destAddr := ADR(aDisanceToStart[nLoopIndex+1]), n := (SIZEOF(aDisanceToStart[0])*(XtsParameterlist.MAX_MOVER_PER_SYSTEM-nLoopIndex-1)));
						aMoversInZone[nLoopIndex] := iMoverPlc;
						aDisanceToStart[nLoopIndex] := lrDistToStart;
						EXIT;
						
					//check next position	
					ELSE 
						;
					END_IF
				END_FOR
			END_IF
		END_IF
	END_WHILE
END_IF
END_METHOD

{attribute 'monitoring':='call'}
PROPERTY StartPositionOnTrack : LREAL
GET
StartPositionOnTrack := _StartPositionOnTrack;
END_GET
SET
_StartPositionOnTrack := StartPositionOnTrack;
END_SET
END_PROPERTY

METHOD Update : HRESULT
VAR

END_VAR
// Nothing todo in Update. Check Prepare
END_METHOD

END_FUNCTION_BLOCK

// COMPENENTs/Zone/I_XTS_Zone
INTERFACE I_XTS_Zone

{attribute 'monitoring':='call'}
PROPERTY CtsMoversInZone : UINT
GET
END_GET
END_PROPERTY

{attribute 'monitoring':='call'}
PROPERTY EndPositionOnTrack : LREAL
GET
END_GET
SET
END_SET
END_PROPERTY

{attribute 'monitoring':='call'}
PROPERTY HR : HRESULT
GET
END_GET
END_PROPERTY

PROPERTY ListOfMoversToCheck : I_CH_List
SET
END_SET
END_PROPERTY

{attribute 'monitoring':='call'}
PROPERTY MoversInZone : REFERENCE TO ARRAY [0..(XtsParameterlist.MAX_MOVER_PER_SYSTEM-1)] OF I_XTS_Mover_PLC
GET
END_GET
END_PROPERTY

{attribute 'monitoring':='call'}
PROPERTY StartPositionOnTrack : LREAL
GET
END_GET
SET
END_SET
END_PROPERTY

END_INTERFACE

// FUNCTIONs/FUN_GetDistToPosModulo
FUNCTION FUN_GetDistToPosModulo : LREAL //This is only working in Positiv Direktion
VAR_INPUT
	TargedPosition : LREAL;
	ActualPosition : LREAL;
	Modulo : LREAL;
END_VAR

VAR
	
END_VAR

IF TargedPosition < ActualPosition THEN
	TargedPosition := TargedPosition + Modulo;
END_IF

FUN_GetDistToPosModulo := TargedPosition - ActualPosition;

END_FUNCTION

// FUNCTIONs/FUN_BuildLogString
FUNCTION FUN_BuildLogString : String
VAR_INPUT
	Pos : LREAL;
	Velocity : LREAL;
	Gap : LREAL;
END_VAR
VAR
	sTemp: STRING;
END_VAR

sTemp := 				CONCAT('Pos:' , LREAL_TO_STRING(Pos));
sTemp := CONCAT(sTemp, 	CONCAT(', Velocity:' , LREAL_TO_STRING(Velocity)));
sTemp := CONCAT(sTemp, 	CONCAT(', Gap:' , LREAL_TO_STRING(Gap)));

FUN_BuildLogString := sTemp;

END_FUNCTION

// COMPENENTs/System/FB_XTS_System
{attribute 'no_explicit_call' := 'Do not call the body - Stick to OOP'}
FUNCTION_BLOCK FB_XTS_System EXTENDS FB_CH_Object IMPLEMENTS I_XTS_System_Registration, I_XTS_System_PLC
VAR	
	{attribute 'hide'}
	bInitDone : BOOL;
	{attribute 'hide'}
    fbMovers     : FB_CH_List;
	{attribute 'hide'}	
	fbStations 	 : FB_CH_List;
	{attribute 'hide'}	
	fbZone 	 : FB_CH_List;
	{attribute 'hide'}	
	fbTrigger 	 : FB_CH_List;
	{attribute 'hide'}	
	iGroup		 : I_XTS_Group;
	{attribute 'hide'}	
    iEnvironment : I_XTS_Environment;
	{attribute 'hide'}
    nState_SEQ_Enabling  : UINT;
	{attribute 'hide'}	
    nState_SEQ_Disabling  : UINT;

	
	fbFeedback : FB_CH_Feedback;
END_VAR

METHOD Disable : CHALET_BaseComponents.I_CH_Feedback
//Disable is allways posible

THIS^.nState_SEQ_Disabling 	:= 1;
THIS^.nState_SEQ_Enabling 	:= 0;

THIS^.SuppressAllDynamicsChanges := TRUE;	

THIS^.fbFeedback.LastCommandAccepted:= TRUE;
THIS^.fbFeedback.ActiveCommand 		:= 'Disable';
THIS^.fbFeedback.Busy 				:= TRUE;	
Disable := THIS^.fbFeedback;
END_METHOD

{attribute 'monitoring':='call'}
PROPERTY Disabled : BOOL
GET
Disabled := nState_SEQ_Disabling = 999 OR 
			(nState_SEQ_Disabling = 0 AND nState_SEQ_Enabling = 0);
END_GET
END_PROPERTY

METHOD PROTECTED Disabling : HRESULT
VAR
	hr : HRESULT;
	bOk : BOOL := TRUE;
	iTempMover : I_XTS_Mover;
END_VAR

VAR_INST
	fbTimeWait : TON; 
	lastHresult : HRESULT;
END_VAR
Disabling := S_PENDING;
CASE nState_SEQ_Disabling OF
	0: // Idle
		Disabling := S_OK;
		
		
	1: // Halt movers
		THIS^.fbMovers.ResetIterator();
		WHILE THIS^.fbMovers.HasNextObject() DO
			IF ToMover(THIS^.fbMovers.GetNextObject(),iTempMover) THEN
				IF iTempMover.MoverInGroup THEN
					hr := GetMostSignificant(hr, iTempMover.HaltCA());
				END_IF
			END_IF
		END_WHILE
		
		IF CheckOk(hr) THEN 
			nState_SEQ_Disabling := 20;
		END_IF	
	
		
	20: // Halting movers	
		THIS^.fbMovers.ResetIterator();
		WHILE THIS^.fbMovers.HasNextObject() DO
			IF ToMover(THIS^.fbMovers.GetNextObject(),iTempMover) THEN
				bOk := bOk AND iTempMover.getAxisRef.NcToPlc.SetVelo = 0;
			END_IF
		END_WHILE
		
		IF bOk THEN 
			nState_SEQ_Disabling := 25;
		END_IF	
		
		
	25: // wait for halt done
		IF iGroup.AllAxesStanding THEN
			nState_SEQ_Disabling := 30;
		END_IF
					
		
	30: // Reset movers
		THIS^.fbMovers.ResetIterator();
		WHILE THIS^.fbMovers.HasNextObject() DO
			IF ToMover(THIS^.fbMovers.GetNextObject(),iTempMover) THEN
				hr := GetMostSignificant(hr, iTempMover.Reset());
			END_IF
		END_WHILE
		
		IF CheckOk(hr) THEN 
			nState_SEQ_Disabling := 40;
		ELSE
			nState_SEQ_Disabling := 1000 + nState_SEQ_Disabling;
		END_IF				
		
		
	40: // Resetting movers
		THIS^.fbMovers.ResetIterator();
		WHILE THIS^.fbMovers.HasNextObject() DO
			IF ToMover(THIS^.fbMovers.GetNextObject(),iTempMover) THEN
				hr := GetMostSignificant(hr, iTempMover.Feedback.HR);
			END_IF
		END_WHILE
		
		IF CheckOk(hr) THEN 
			nState_SEQ_Disabling := 63;
		ELSIF FAILED(hr) THEN
			nState_SEQ_Disabling := 1000 + nState_SEQ_Disabling;
		END_IF
	
		
	63: // Reset group
		hr :=  iGroup.Reset();
		
		IF CheckOk(hr) THEN 
			nState_SEQ_Disabling := 64;
		ELSE
			nState_SEQ_Disabling := 1000 + nState_SEQ_Disabling;
		END_IF		
		
		
	64: // Resetting group
		hr := iGroup.HR;
		
		IF CheckOk(hr) THEN 
			nState_SEQ_Disabling := 70;
		ELSIF FAILED(hr) THEN
			nState_SEQ_Disabling := 1000 + nState_SEQ_Disabling;
		END_IF		
		
		
	70: // Disable group
		hr := iGroup.Disable();
		
		IF CheckOk(hr) THEN 
			nState_SEQ_Disabling := 100;
		ELSE
			nState_SEQ_Disabling := 1000 + nState_SEQ_Disabling;
		END_IF	
		
		
   100: // Disabling group
		hr := iGroup.HR;
		
		IF CheckOk(hr) THEN 
			nState_SEQ_Disabling := 110;
		ELSIF FAILED(hr) THEN
			nState_SEQ_Disabling := 1000 + nState_SEQ_Disabling;
		END_IF			
		
		
	110: // Remove movers from group
		hr := iGroup.UngroupAllAxes();
		
		IF CheckOk(hr) THEN 
			nState_SEQ_Disabling := 120;
		ELSE
			nState_SEQ_Disabling := 1000 + nState_SEQ_Disabling;
		END_IF		
	
		
	120: // Removing movers from group
		hr := iGroup.HR;
		
		IF CheckOk(hr) THEN 
			nState_SEQ_Disabling := 130;
		ELSIF FAILED(hr) THEN
			nState_SEQ_Disabling := 1000 + nState_SEQ_Disabling;
		END_IF	

		
	130: // write state to movers
		THIS^.fbMovers.ResetIterator();
		WHILE THIS^.fbMovers.HasNextObject() DO
			IF ToMover(THIS^.fbMovers.GetNextObject(),iTempMover) THEN
				iTempMover.MoverInGroup := FALSE;
			END_IF
		END_WHILE

		nState_SEQ_Disabling := 170;	
		
		
	170: // Disable movers
		THIS^.fbMovers.ResetIterator();
		WHILE THIS^.fbMovers.HasNextObject() DO
			IF ToMover(THIS^.fbMovers.GetNextObject(),iTempMover) THEN
				hr := GetMostSignificant(hr, iTempMover.Disable());
			END_IF
		END_WHILE
		
		IF CheckOk(hr) THEN 
			nState_SEQ_Disabling := 180;
		ELSE
			nState_SEQ_Disabling := 1000 + nState_SEQ_Disabling;
		END_IF			
		
		
	180: // Disabling movers
		THIS^.fbMovers.ResetIterator();
		WHILE THIS^.fbMovers.HasNextObject() DO
			IF ToMover(THIS^.fbMovers.GetNextObject(),iTempMover) THEN
				hr := GetMostSignificant(hr, iTempMover.Feedback.HR);
			END_IF
		END_WHILE
		
		IF CheckOk(hr) THEN 
			nState_SEQ_Disabling := 200;
		ELSIF FAILED(hr) THEN
			nState_SEQ_Disabling := 1000 + nState_SEQ_Disabling;
		END_IF		

		
	200: // Wait 1 second according to documentation
		fbTimeWait.IN := TRUE;
		fbTimeWait.PT := T#1S;	
		fbTimeWait();
		
		IF fbTimeWait.Q THEN
			fbTimeWait.IN := FALSE;
			fbTimeWait();
			nState_SEQ_Disabling := 999;
		END_IF
	
		
   999: //Done
   		Disabling := S_OK;

		
	1000..1999://Error
		hr := GetMostSignificant(lastHresult, E_FAIL);	
END_CASE


//store last information
lastHresult := hr;


// Propagate error
IF FAILED(hr) THEN
	Disabling := hr;
END_IF
END_METHOD

METHOD Enable : CHALET_BaseComponents.I_CH_Feedback
IF NOT THIS^.fbFeedback.Done THEN
	//Error active/not ready
	THIS^.fbFeedback.LastCommandAccepted 	:= FALSE;

ELSIF nState_SEQ_Enabling <> 0 THEN
	//System is partial or full enabled. Disable first.
	THIS^.fbFeedback.LastCommandAccepted 	:= FALSE;
ELSE
	
	THIS^.SuppressAllDynamicsChanges := FALSE;	

	THIS^.nState_SEQ_Disabling 	:= 0;
	THIS^.nState_SEQ_Enabling 	:= 1;
	THIS^.fbFeedback.LastCommandAccepted 	:= TRUE;
	THIS^.fbFeedback.ActiveCommand 			:= 'Enable';
	THIS^.fbFeedback.Busy 				 	:= TRUE;	
END_IF

Enable := THIS^.fbFeedback;
END_METHOD

{attribute 'monitoring':='call'}
PROPERTY Enabled : BOOL
GET
Enabled := nState_SEQ_Enabling = 999;
END_GET
END_PROPERTY

METHOD PROTECTED Enabling : HRESULT
VAR
	hr : HRESULT;

	iTempMover : I_XTS_Mover;
END_VAR

VAR_INST
	fbTimeOutSeq : TON; 
	lastHresult : HRESULT;
	nModuleCount : UDINT;
	nLoopCount : UDINT;
END_VAR
Enabling := S_PENDING;
CASE nState_SEQ_Enabling OF
	0: // Idle
		Enabling := S_OK;

	1: // Check OP mode
		IF THIS^.iEnvironment.UtilityEnvirement.XpuTcIo(1).GetOperationMode() = OperationMode.Normal THEN
			nState_SEQ_Enabling := 2; // Check 48V of all Module
		ELSE
			nState_SEQ_Enabling := 3; // in Simulation check of 48V not necessary
		END_IF
		
		
	2: // ToDo: check 48V of all Module?
		nModuleCount:= THIS^.iEnvironment.UtilityEnvirement.XpuTcIo(1).PartTcIo(1).GetModuleCount();
		nState_SEQ_Enabling := 3;
		FOR nLoopCount := 1 TO nModuleCount DO
			IF THIS^.iEnvironment.UtilityEnvirement.XpuTcIo(1).PartTcIo(1).ModuleTcIo(1).GetDCLinkVoltage() < 20 AND
			   THIS^.iEnvironment.UtilityEnvirement.XpuTcIo(1).PartTcIo(1).ModuleTcIo(1).GetDCLinkVoltage() > 56 THEN	
				nState_SEQ_Enabling := 2;				     
			END_IF		
		END_FOR

		
	3: // ask for MoverId Detection Mode	
		IF Environment.UtilityEnvirement.XpuTcIo(1).GetMoverIdDetectionMode() = MoverIdDetectionMode.Standard THEN			
			nState_SEQ_Enabling := 10;
		ELSIF Environment.UtilityEnvirement.XpuTcIo(1).GetMoverIdDetectionMode() = MoverIdDetectionMode.Mover1 THEN
			nState_SEQ_Enabling := 5;
		ELSE // todo: MoverIdDetectionMode.MultipleMover1
			;
		END_IF
		

	5: // Trigger Mover ID dedection 
		IF NOT Environment.UtilityEnvirement.XpuTcIo(1).GetIsMoverIdDetectionActive() AND
		   NOT Environment.UtilityEnvirement.XpuTcIo(1).GetIsMoverIdDetectionValid() THEN
			// Set the Trigger for ID detection
			Environment.UtilityEnvirement.XpuTcIo(1).TriggerMoverIdDetection();
		ELSIF Environment.UtilityEnvirement.XpuTcIo(1).GetIsMoverIdDetectionValid() THEN
			// successful
			nState_SEQ_Enabling := 10;
		ELSIF Environment.UtilityEnvirement.XpuTcIo(1).GetHasMoverIdDetectionError() THEN
			// error
			nState_SEQ_Enabling := 1000 + nState_SEQ_Enabling;
		ELSE 
			; // wait for valid or error					
		END_IF
		
	
	10: // Reset movers
		THIS^.fbMovers.ResetIterator();
		WHILE THIS^.fbMovers.HasNextObject() DO
			IF ToMover(THIS^.fbMovers.GetNextObject(), iTempMover) THEN
				hr := GetMostSignificant(hr, iTempMover.Reset());
			END_IF
		END_WHILE
		
		IF CheckOk(hr) THEN 
			nState_SEQ_Enabling := 20;
		ELSE
			nState_SEQ_Enabling := 1000 + nState_SEQ_Enabling;
		END_IF
		
		
	20: // Resetting movers
		THIS^.fbMovers.ResetIterator();
		WHILE THIS^.fbMovers.HasNextObject() DO
			IF toMover(THIS^.fbMovers.GetNextObject(), iTempMover) THEN
				hr := GetMostSignificant(hr, iTempMover.Feedback.HR);
			END_IF
		END_WHILE
		
